*)
VAR CONSTANT
	(*Costant in lux obj*)
	NO_DIMMING	: BYTE:=0;
	DIMMING		: BYTE:=1;
	ROT			: BOOL:=1;
	GRUN		: BOOL:=0;
END_VAR

VAR_INPUT
	(* Settings *)
	ID					: WORD;
	DimmingType		: BYTE;	 (* /0: no dimming (digital), 1: dimming (analog) *)
	DimmingValForTimer	: INT;	 (* /valore 0...100 del dimming di default del lux sotto timer *)
	(* Controls *)
	CTRL_MODE			: en_Modality;	 (* 0:MAN OFF, 1:MAN-ON, 3:Timer laser, 2:Cronografo*)
	CTRL_MODE_BackUp	: en_Modality;	 (*Salvo il valore di default per il ripristino *)
	LuxTimer		: TIME; (* Tempo di accensione del lux settato nella tabella TabLuxPsg ottenuta dal file di config su SD *)
	HourMinStartOn	: TOD; (* Orario di start per rilevazione sensori start timer (Mode 03) *)
	HourMinEndOn	: TOD; (* Orario di end per rilevazione sensori start timer (Mode 03) *)
	ValInCronoInLux : INT;	(* Valore del setpoint arrivato dal crono *)
	RefTableAutLuxPsg : WORD; (* indice di riferimento alla tabella AUT_LUX_PSG se mode = 3 *)
	RestoreKey		: BOOL; (* se attivato viene ripristinato il mode di default *)
	CtrlTrig		: BOOL; (* Trigger for timer start *)
	CtrlKeyList		: ARRAY [0..9] OF BOOL; (* External KEY control input *)
	KeyQty			: BYTE; (* numero di key all'ingresso *)
	KeyMode			: en_KeyMode;	(* BYTE; //Modalità di funzionamento richiesta dal key *)
	DimmingValForKeyList: ARRAY [0..9] OF INT;
	DimmingValForKeyMax: BOOL; (* Se TRUE --> si sceglie il valore massimo; Se FALSE --> si sceglie il valore minimo *)
	ActionKey		: en_ActionKey; (* 00-NormalMode, 01-SwitchON, 02-SwitchOFF, 03-Restore *)
	(* Physical inputs *)
	Lux_State		: BOOL; (* Status feedback *)
	Lux_StateAnalog	: WORD;  (* feedback analogico dal campo GIURE ver 008  *)

END_VAR
VAR_IN_OUT
	LocalWorkingTime		: DWORD; (* [sec] Internal working time counter *)
	LocalPowerOnCycles		: WORD;	(* DWORD; Internal counter of power-on cycles *)
	LocalEnergyCounter		: WORD;	(* DWORD;  [E-1 kWh] Internal energy counter *)
	LocalEnergyCounter_t 	: DWORD; (* Temporary energy in E-2*Wsec *)
END_VAR
VAR_OUTPUT
	(* Physical outputs *)
	LuxDigitalOut	: BOOL;
	LuxAnalogOut	: WORD;
	LuxTypeOut		: BOOL;
	Lux_Enable		: BOOL;	(*  uscita logica per compatibilità con sw preesistente (ex (* Control output *)) *)
	Lux_EnableAnalog : WORD;
	(* Status *)
	Status_Log		: BYTE;
	Status_Vis 		: DWORD;
END_VAR
VAR
	TickTimer		: TON := ( PT:=T#1S );
	TrigTimer		: TOF ;

	KeyTimer		: TIME := T#200ms;
	sLux_EN			: FLT_EVENT;
	chkLux_ST		: FLT_TIME := ( TTAP:=T#20S, INITEV:=FALSE );
	chkLux_ST_Analog: FLT_TIME := ( TTAP:=T#20S, INITEV:=FALSE );
	HourMinNow		: STRING;
	semaphore		: BOOL:=GRUN;
	OnFromKey		: BOOL;
	fTrigFun		: F_TRIG;
	rTrigFun		: R_TRIG;
	fTrigKey		: F_TRIG;
	ActionKeyState	: en_ActionKey;
	KeyCounter, x	: BYTE;
	CtrlKey			: BOOL;
	DimmingValForKey: INT; (* valore 0...100 del dimming di default del lux sotto key *)
	ModeToServer : BYTE;
	ForcedOn : BYTE;
	ForcedOff : BYTE;

END_VAR
(* Con l'ID si identifica il numero del lux sul campo quindi il suo valore può variare da 1 a LUXM_MAX (attualmente 1...900) *)
IF (KeyMode = BUTTON_NO) OR (KeyMode = BUTTON_NC) THEN (* se si usano dei pulsanti sui vari digital input...*)
	KeyCounter := 0;
	FOR x:=0 TO  KeyQty-1 DO
		IF CtrlKeyList[x] = 1 THEN
			KeyCounter := KeyCounter + 1;
		END_IF
	END_FOR
	IF (KeyCounter MOD 2) = 0 THEN
		CtrlKey := FALSE;
	ELSE
		DimmingValForKey := DimmingValForKeyList[0]; (* In caso di pulsanti si prende il valore della posizione 0 dell'array *)
		CtrlKey := TRUE;
	END_IF
ELSE (* altrimenti se uso l'interruttore ne posso usare solo 1 nella posizione 0 dell'array *)
	IF (DimmingValForKeyMax) THEN
		DimmingValForKey := 0;
		FOR x:=0 TO  KeyQty-1 DO
			IF (CtrlKeyList[x] = 1) AND (DimmingValForKeyList[x] > DimmingValForKey)
			THEN
				DimmingValForKey := DimmingValForKeyList[x];
			END_IF
		END_FOR
	ELSIF NOT(DimmingValForKeyMax) THEN
		DimmingValForKey :=1000;
		FOR x:=0 TO  KeyQty-1 DO
			IF (CtrlKeyList[x] = 1) AND (DimmingValForKeyList[x] < DimmingValForKey)
			THEN
				DimmingValForKey := DimmingValForKeyList[x];
			END_IF
		END_FOR
	END_IF
	CtrlKey := 0;
	FOR x:=0 TO  KeyQty-1 DO
			CtrlKey := CtrlKey OR CtrlKeyList[x];
	END_FOR

END_IF

CASE DimmingType OF (* set dell' AsiTypeOut per sapere se eseguire il set di un analog out o di un digital out *)
	NO_DIMMING:	(* if no dimming we are using a digital output *)
		LuxTypeOut := DIGITAL; (* Set digital out mode *)
	DIMMING:	(*  if dimming we are using analog output *)
		LuxTypeOut := ANALOG; (* Set analog out mode *)
END_CASE

(* Control logic *)
(* Restore mode and value	*)
IF RestoreKey THEN
	CTRL_MODE := CTRL_MODE_BackUp;
END_IF

CASE CTRL_MODE OF
	ManualeOff: (*  0 Manuale Off *)
		(* Se commutazione arrivata da key durante funzionamento in timer o cronografo *)
		IF  NOT(CtrlKey) AND (ActionKey > NormalMode) AND ( ActionKeyState = SwitchOFF)THEN
			ActionKeyState := NormalMode;
			CTRL_MODE := CTRL_MODE_BackUp;
		ELSE
			CASE DimmingType OF
				NO_DIMMING:	(* if no dimming we are using a digital output *)
					LuxDigitalOut := TRUE; (* Lux spento (digital) *)
				DIMMING:	(*  if dimming we are using analog and digital output *)
					DimmerCtrl(); (* In caso di switch off in manuale è sempre zero anche se arriva da key *)
			END_CASE
		END_IF
	ManualeOn: (*  1 Manuale On *)
		(* Se commutazione arrivata da key durante funzionamento in timer o cronografo *)
		IF  NOT(CtrlKey) AND (ActionKey > NormalMode) AND ( ActionKeyState = SwitchON) THEN
			ActionKeyState := NormalMode;
			CTRL_MODE := CTRL_MODE_BackUp;
		ELSE
			CASE DimmingType OF
				NO_DIMMING:	(* if no dimming we are using a digital output *)
					LuxDigitalOut := FALSE; (* Lux acceso (digital) *)
				DIMMING:	(*  if dimming we are using analog and digital output  *)
					IF ActionKeyState = SwitchON THEN
						DimmerCtrlKeyOn(); (* Se il manuale on è settato a causa di un key si impongono i dati del key stesso *)
					ELSE
						DimmerCtrl();
					END_IF
			END_CASE
		END_IF
	Cronografo: (*  2 Cronografo *)
		IF  (CtrlKey) AND (ActionKey > NormalMode) THEN
			CASE  ActionKey OF
				SwitchON: 	(* Corrisponde al manuale ON *)
					CTRL_MODE := ManualeOn;
					ActionKeyState := SwitchON;
					CASE DimmingType OF
						NO_DIMMING:	(* if no dimming we are using a digital output *)
							LuxDigitalOut := FALSE; (* Lux acceso (digital) *)
						DIMMING:	(*  if dimming we are using analog and digital output  *)
							DimmerCtrlKeyOn();
					END_CASE

				SwitchOFF:	(* Corrisponde al manuale OFF  *)
					CTRL_MODE := ManualeOff;
					ActionKeyState := SwitchOFF;
					CASE DimmingType OF
						NO_DIMMING:	(* if no dimming we are using a digital output  *)
							LuxDigitalOut := TRUE; (* Lux spento (digital)  *)
						DIMMING:	(*  if dimming we are using analog and digital output  *)
							DimmerCtrlKeyOff();
					END_CASE
			END_CASE
		ELSE
			CASE DimmingType OF
				NO_DIMMING:	(* if no dimming we are using a digital output  *)
					IF ValInCronoInLux = 1000 (* OR ( LuxElement[i].PressKeyVisuOn)  *)
						THEN
						LuxDigitalOut := FALSE; (* Lux acceso (digital)  *)
						ELSE IF ValInCronoInLux = 0 (* OR ( NOT LuxElement[i].PressKeyVisuOn)  *)
							THEN
							LuxDigitalOut := TRUE; (* Lux spento (digital)  *)
						END_IF
					END_IF
				DIMMING:	(*  if dimming we are using analog output  *)
					DimmerCtrl();
			END_CASE
		END_IF
	Timer: (*  3 Timer   *)
	IF  (CtrlKey) AND (ActionKey > NormalMode) THEN
		CASE  ActionKey OF
			SwitchON: 	(* Corrisponde al manuale ON  *)
				CTRL_MODE := ManualeOn;
				ActionKeyState := SwitchON;
				CASE DimmingType OF
					NO_DIMMING:	(* if no dimming we are using a digital output  *)
						LuxDigitalOut := FALSE; (* Lux acceso (digital)  *)
					DIMMING:	(*  if dimming we are using analog and digital output   *)
						DimmerCtrlKeyOn();
				END_CASE

			SwitchOFF:	(* Corrisponde al manuale OFF  *)
				CTRL_MODE := ManualeOff;
				ActionKeyState := SwitchOFF;
				CASE DimmingType OF
					NO_DIMMING:	(* if no dimming we are using a digital output  *)
						LuxDigitalOut := TRUE; (* Lux spento (digital)  *)
					DIMMING:	(*  if dimming we are using analog and digital output  *)
						DimmerCtrlKeyOff();
				END_CASE
		END_CASE
	ELSE
		CASE DimmingType OF
			NO_DIMMING:	(* if no dimming we are using a digital output  *)
				HourMinNow:=CONCAT('TOD#', BYTE_TO_STRING(Sys.Time_Hour));
				HourMinNow:=CONCAT(HourMinNow, ':');
				HourMinNow:=CONCAT(HourMinNow, BYTE_TO_STRING(Sys.Time_Min));
				HourMinNow:=CONCAT(HourMinNow,':00');

				(* Trig timer *)
				TrigTimer.PT:=LuxTimer;
				TrigTimer(IN:= CtrlTrig);

				IF (((STRING_TO_TOD(HourMinNow) > HourMinStartOn) AND (STRING_TO_TOD(HourMinNow) < HourMinEndOn))  (* Se siamo nell'orario corretto  *)
				OR ((LuxDigitalOut = FALSE) AND (TrigTimer.Q = FALSE))) (* oppure si era acceso e adesso siamo passati fuori orario e dobbiamo spegnere  *)
				THEN
					IF TrigTimer.Q THEN
						LuxDigitalOut := FALSE; (* Lux acceso (digital)  *)
						ELSE
							LuxDigitalOut:= TRUE; (* Lux spento (digital)  *)
					END_IF
				END_IF
			DIMMING:	(*  if dimming we are using analog output  *)

				HourMinNow:=CONCAT('TOD#', BYTE_TO_STRING(Sys.Time_Hour));
				HourMinNow:=CONCAT(HourMinNow, ':');
				HourMinNow:=CONCAT(HourMinNow, BYTE_TO_STRING(Sys.Time_Min));
				HourMinNow:=CONCAT(HourMinNow,':00');

				(* Trig timer *)
				TrigTimer.PT:=LuxTimer;
				TrigTimer(IN:= CtrlTrig);

				IF (((STRING_TO_TOD(HourMinNow) > HourMinStartOn) AND (STRING_TO_TOD(HourMinNow) < HourMinEndOn))  (* Se siamo nell'orario corretto  *)
				OR ((LuxDigitalOut = FALSE) AND (TrigTimer.Q = FALSE))) (* oppure si era acceso e adesso siamo passati fuori orario e dobbiamo spegnere  *)
				THEN
					IF TrigTimer.Q THEN
						DimmerCtrl(); (* Lux acceso  *)
						ELSE
							LuxAnalogOut := 0; (* Lux spento  *)
							LuxDigitalOut := TRUE; (* Lux spento (digital)  *)
					END_IF
				END_IF
		END_CASE
		END_IF
	KeyControl: (*  4 Key function  *)
		IF CtrlKey THEN
			CASE DimmingType OF
				NO_DIMMING:	(* if no dimming we are using a digital output  *)
					LuxDigitalOut := FALSE; (* Lux acceso (digital)  *)
				DIMMING:	(*  if dimming we are using analog and digital output   *)
					DimmerCtrlKeyOn();
			END_CASE
		ELSIF CtrlKey = 0 THEN
			CASE DimmingType OF
				NO_DIMMING:	(* if no dimming we are using a digital output  *)
					LuxDigitalOut := TRUE; (* Lux spento (digital)  *)
				DIMMING:	(*  if dimming we are using analog and digital output  *)
					DimmerCtrlKeyOff();
			END_CASE
		END_IF
	END_CASE

(* ----------------------------------------------------------------------------------------------------------------------------------------  *)
(* Se i pin del feedback relè non sono cavallottati si usa la seguente riga al posto di quelle successive indicate da(#)  *)
(* REL_ST := LUX_ST[ID];	  																					 *)
(* ----------------------------------------------------------------------------------------------------------------------------------------   *)

(* setting della variabile REL_EN per compatibilità con il sw preesistente  *)
CASE DimmingType OF
	NO_DIMMING:	(* if no dimming we are using a digital output  *)
	IF LuxDigitalOut = TRUE  (* Lux spento  *)
		THEN
			(* Lux_State := FALSE;	//A causa del cavallotto sui pin del relè forzo a falso (#)  *)
			(* Lux_State := LUX_ST[ID];	  *)
			Lux_Enable := FALSE;
		ELSIF LuxDigitalOut = FALSE  (* Lux acceso			   *)
			THEN
				(* Lux_State := LUX_ST[ID];	//Quando so che la luce è accesa leggo lo stato del pin (che essendo cavallottato sarà a 1) (#)  *)
				Lux_Enable := TRUE;
	END_IF

	DIMMING:	(*  if dimming we are using analog output  *)
	IF LuxAnalogOut  = 0 (* Lux spento				  *)
		THEN
			(* REL_ST := FALSE;	 A causa del cavallotto sui pin del relè forzo a falso (#)  *)
			(* Lux_State := LUX_ST[ID];	  *)
			Lux_State:= TRUE;	(* aggiunta perchè non ho feedback sul relè *)
			Lux_Enable := FALSE;
			Lux_EnableAnalog := LuxAnalogOut; (* GIURE ver 008   *)
		ELSIF LuxAnalogOut > 0  (* Lux acceso			  *)
			THEN
				(* Lux_State := LUX_ST[ID];	 Quando so che la luce è accesa leggo lo stato del pin (che essendo cavallottato sarà a 1) (#)  *)
				Lux_State:= TRUE; (* aggiunta perchè non ho feedback sul relè *)
				Lux_Enable := TRUE;
				Lux_EnableAnalog := LuxAnalogOut;  (* GIURE ver 008  *)
	END_IF

END_CASE
(* Temporary energy counter *)
TickTimer(IN:=NOT TickTimer.Q);
IF TickTimer.Q AND Lux_Enable THEN
	LocalWorkingTime:=LocalWorkingTime+1;
	IF LocalEnergyCounter_t>36000000 THEN
		LocalEnergyCounter_t:=LocalEnergyCounter_t-36000000;
		LocalEnergyCounter:=LocalEnergyCounter+1;
	END_IF
END_IF

(* Generate status events *)
sLux_EN(IN:=Lux_Enable);
IF sLux_EN.EVL THEN
	LogEv(EL_Log,EO_LUX,ID,2,'Light OFF'); (* Light OFF  *)
END_IF
IF sLux_EN.EVH THEN
	LogEv(EL_Log,EO_LUX,ID,3,'Light ON'); (* Light ON  *)
	LocalPowerOnCycles:=LocalPowerOnCycles+1;
END_IF


(* Check status feedback *) (* GIURE ver 008 - aggiunta controllo valori analogici  *)
chkLux_ST_Analog(IN:=(Lux_StateAnalog<>Lux_EnableAnalog));
IF chkLux_ST_Analog.EVH THEN
	LogEv(EL_Alarm,EO_LUX,ID,9,'Fail Analog');(*  Feedback failure - Lux_StateAnalog<>Lux_EnableAnalog*)
END_IF
IF chkLux_ST_Analog.EVL THEN
	LogEv(EL_Log,EO_LUX,ID,1,'Successful Analog'); (*  Light feedback OK - Lux_StateAnalog = Lux_EnableAnalog  *)
END_IF
(* Check status feedback *)
chkLux_ST(IN:=(Lux_State<>Lux_Enable));
IF chkLux_ST.EVH THEN
	LogEv(EL_Alarm,EO_LUX,ID,9,'Fail'); (*  Feedback failure - Lux_State<>Lux_Enable  *)
END_IF
IF chkLux_ST.EVL THEN
	LogEv(EL_Log,EO_LUX,ID,1,'Successful'); (*  Light feedback OK - Lux_State = Lux_Enable  *)
END_IF


(* Status color *)
IF chkLux_ST.OUT THEN
	Status_Log:=2; Status_Vis:=COLOR_RED;
ELSE
	Status_Log:=0;
	Status_Vis:=SEL(Lux_Enable,COLOR_GREEN_OFF,COLOR_GREEN);
END_IF

(* Salvataggio dati in array ordinato per numero di ID utile per la visualizzazione  *)
DataLuxForVis[ID].VisStatus:=Status_Vis;
DataLuxForVis[ID].VisTimer:=LuxTimer/1000;
DataLuxForVis[ID].VisMod:=CTRL_MODE;
(* DataLuxForVis[ID].VisMod:=any_num_to_byte(CTRL_MODE); *)
END_FUNCTION_BLOCK
ACTION AddLogData:
Logger.s1:=INSERT('&LUX=',WORD_TO_STRING(ID),4);
IF ID<10 THEN Logger.s1:=INSERT(Logger.s1,'0',4); END_IF

Logger.s1:=CONCAT(Logger.s1,BOOL_TO_STRING(Lux_Enable));				Logger.s1:=CONCAT(Logger.s1,';');
Logger.s1:=CONCAT(Logger.s1,DWORD_TO_STRING(LocalWorkingTime));		Logger.s1:=CONCAT(Logger.s1,';');
Logger.s1:=CONCAT(Logger.s1,DWORD_TO_STRING(LocalPowerOnCycles));	Logger.s1:=CONCAT(Logger.s1,';');

CASE CTRL_MODE OF		(* modifica GIURE 009 ver 1.3 *)
	0: 	(*  Manuale OFF *)
		ModeToServer := 0;
		ForcedOn := 0;
		ForcedOff := 1;
	1:	(*  Manuale ON *)
		ModeToServer := 1;
		ForcedOn := 1;
		ForcedOff := 0;
	2:	(*  Cronografo *)
		ModeToServer := 2;
		ForcedOn := 0;
		ForcedOff := 0;
	3: 	(* Timer *)
		ModeToServer := 3;
		ForcedOn := 0;
		ForcedOff := 0;
END_CASE
Logger.s1:=CONCAT(Logger.s1,BYTE_TO_STRING(ModeToServer));			Logger.s1:=CONCAT(Logger.s1,';');
Logger.s1:=CONCAT(Logger.s1,BYTE_TO_STRING(Status_Log));				Logger.s1:=CONCAT(Logger.s1,';');
Logger.s1:=CONCAT(Logger.s1,BYTE_TO_STRING(ForcedOn));				Logger.s1:=CONCAT(Logger.s1,';');
Logger.s1:=CONCAT(Logger.s1,BYTE_TO_STRING(ForcedOff));				Logger.s1:=CONCAT(Logger.s1,';');
Logger.s1:=CONCAT(Logger.s1,BYTE_TO_STRING(DimmingType));			Logger.s1:=CONCAT(Logger.s1,';');
Logger.s1:=CONCAT(Logger.s1,WORD_TO_STRING(Lux_EnableAnalog/100));

ADDSTRING(ADR(Logger.TData), ADR(Logger.s1), Logger.TLen);
END_ACTION
ACTION DimmerCtrl:
CASE CTRL_MODE OF
	0: (* Manuale Off *)
		LuxAnalogOut := 0; (* Lux spento *)
		LuxDigitalOut := TRUE; (* Lux spento (digital) *)
	1: (* Manuale On *)
		LuxAnalogOut := 10000; (* Lux acceso *)
		LuxDigitalOut := FALSE; (* Lux acceso (digital) *)
	2: (* Cronografo *)
		IF ValInCronoInLux > 0 THEN
			LuxDigitalOut := FALSE; (* Lux acceso (digital) *)
			ELSE
				LuxDigitalOut := TRUE; (* Lux spento (digital) *)
		END_IF
		LuxAnalogOut := INT_TO_WORD(ValInCronoInLux*10);
	3: (* Timer 		 *)
		IF DimmingValForTimer > 0 THEN
			LuxDigitalOut := FALSE; (* Lux acceso (digital) *)
			ELSE
				LuxDigitalOut := TRUE; (* Lux spento (digital) *)
		END_IF
		LuxAnalogOut := INT_TO_WORD(DimmingValForTimer*10);
	ELSE (* default *)
		LuxDigitalOut := FALSE; (* Lux acceso (digital) *)
		LuxAnalogOut := 10000;
END_CASE
END_ACTION
ACTION DimmerCtrlKeyOff:
LuxAnalogOut := 0; (*/Lux spento*)
LuxDigitalOut := TRUE; (*Lux spento (digital)*)
END_ACTION
ACTION DimmerCtrlKeyOn:
LuxAnalogOut := INT_TO_WORD(DimmingValForKey*10);
LuxDigitalOut := FALSE; (*Lux acceso (digital) *)
END_ACTION
ACTION StatReset:
(* Reset statistic counters *)
LocalWorkingTime:=0;
LocalPowerOnCycles:=0;
LocalEnergyCounter:=0;
END_ACTION

(* POU Plant_Objects/obj_TPV, ST *)
FUNCTION_BLOCK obj_TPV
(* === TEMPERATURE PROBE  ===
   v1.0[16/04/15] - Versioning
*)
VAR CONSTANT
	NormalEv		: BYTE := 0;
	ErrorEv			: BYTE := 1;
	WarningEv		: BYTE := 2;
END_VAR
VAR_INPUT
	(* Settings *)
	ID				: BYTE;
	TAP				: BYTE:=4;	   (* Consecutive checks filter *)
	INITEV			: BOOL:= TRUE; (* Generate init OK event *)
	IN_EMIN			: INT :=-2000; (* Low error limit *)
	IN_WMIN			: INT := -550; (* Low warning value *)
	IN_WMAX			: INT :=  900; (* High warning value *)
	IN_EMAX			: INT := 8500; (* High error limit *)
	ERR_MIN_SHORT	: BOOL:= TRUE; (* TRUE  ==> EMIN=Short        , EMAX=Disconnected
									  FALSE ==> EMIN=Disconnected , EMAX=Short 		 *)
	(* Physical input *)
	IN			: INT;
END_VAR
VAR_OUTPUT
	WRN			: BOOL;	(* Value in warning range *)
	ERR			: BOOL;	(* Value error *)
	HI			: INT;	(* Highest value - cleared by Stat_Reset() action *)
	AVG			: INT; 	(* Average value - updated by Mean() action, cleared by Mean_Reset() action *)
	LOW			: INT;	(* Lowest value  - cleared by Stat_Reset() action *)

	Status_Log	: WORD;
	Status_Vis	: DWORD;
END_VAR
VAR
	cnt			: BYTE;
	event		: BYTE := 0;	(* 0: monitoring a generic, 1: monitoring an error, 2: monitoring a warning *)
	asum		: DINT;
	acnt		: WORD;
END_VAR
(* Check probe value limits *)
IF IN<=IN_EMIN OR IN>=IN_EMAX THEN
	IF NOT ERR THEN
		IF event <> ErrorEv THEN
			cnt := 1;
			event := ErrorEv;
		ELSE
			cnt:=cnt+1;
		END_IF

		IF cnt>TAP THEN
			cnt:=0;
			ERR:=TRUE; WRN:=FALSE;
			IF ( ERR_MIN_SHORT=TRUE  AND IN<=IN_EMIN ) OR ( ERR_MIN_SHORT=FALSE AND IN>=IN_EMAX ) THEN
				LogEv(EL_Alarm,EO_TPV,ID,5,INT_TO_STRING(IN));
			ELSE
				LogEv(EL_Alarm,EO_TPV,ID,4,INT_TO_STRING(IN));
			END_IF
		END_IF
	END_IF
ELSIF IN<=IN_WMIN OR IN>=IN_WMAX THEN
	IF NOT WRN THEN
		IF event <> WarningEv THEN
			cnt := 1;
			event := WarningEv;
		ELSE
			cnt:=cnt+1;
		END_IF

		IF cnt>TAP THEN
			cnt:=0;
			ERR:=FALSE; WRN:=TRUE;
			LogEv(EL_Wrn,EO_TPV,ID,SEL(IN<=IN_WMIN,3,2),INT_TO_STRING(IN));
		END_IF
	END_IF
ELSE
	IF INITEV OR WRN OR ERR THEN
		IF event <> NormalEv THEN
			cnt := 1;
			event := NormalEv;
		ELSE
			cnt:=cnt+1;
		END_IF

		IF cnt>TAP THEN
			cnt:=0;
			INITEV:=FALSE; ERR:=FALSE; WRN:=FALSE;
			LogEv(EL_Log,EO_TPV,ID,1,'Probe_OK');
		END_IF
	END_IF
END_IF


(*
(* Average value *)
IF acnt>=500 THEN
	Mean();
	asum := asum - AVG;
	acnt := acnt - 1;
END_IF

asum := asum + IN;
acnt := acnt + 1;
*)

AVG := IN;



(* Statistics values *)
IF IN<LOW THEN LOW:=IN; END_IF
IF IN>HI  THEN HI :=IN; END_IF

Lamp.obj_Status := Status_Log;
Lamp.UpdateStatus();

(* Status Log *)
IF ERR THEN	Status_Log := 2; Status_Vis := COLOR_RED;
ELSIF WRN THEN Status_Log := 1;	Status_Vis := COLOR_YELLOW;
ELSE Status_Log := 0; Status_Vis := COLOR_GREEN;
END_IF
END_FUNCTION_BLOCK
ACTION AddLogData:
Logger.s1:=INSERT('&TPV=',BYTE_TO_STRING(ID),4);
IF ID<10 THEN Logger.s1:=INSERT(Logger.s1,'0',4); END_IF
(*
Mean();
*)
Logger.s1:=CONCAT(Logger.s1,INT_TO_STRING(AVG));		Logger.s1:=CONCAT(Logger.s1,';');

Logger.s1:=CONCAT(Logger.s1,WORD_TO_STRING(Status_Log));
ADDSTRING(ADR(Logger.TData), ADR(Logger.s1), Logger.TLen);
END_ACTION
ACTION Mean:
(*AVG := DINT_TO_INT(asum/acnt); *)


AVG := IN;
END_ACTION
ACTION Mean_Reset:
AVG:=IN;
asum:=IN;
acnt:=1;
END_ACTION
ACTION Stat_Reset:
HI:=IN;
LOW:=IN;
END_ACTION

(* POU Plant_Objects/obj_VRD_new, ST *)
FUNCTION_BLOCK obj_VRD_new
(* === VALVOLA RIPARTITORE ===
   v1.0[16/04/15] - Versioning
*)
VAR CONSTANT
	Chk_CntSecAlarm	: INT := 900;	(* 900s = 15 minutes -> Observation itme *)
END_VAR
VAR_INPUT
	(* Settings *)
	ID				: BYTE;
	(* Controls *)
	RUN  			: BOOL;					(* Control input *)
	ReducedRange	: BOOL := FALSE;		(* If true output value is among 2 and 10V, otherwise 0-10V *)

	(* Physical inputs *)
	TEMP 			: INT;		(* Input temperature from sensor *)
	STATUS 			: WORD;		(* Input position from valve *)

	InitOK			: BOOL;
	Alarm1			: BOOL;
	Alarm2			: BOOL;
	Warning			: BOOL;

	Ctrl_Init		: BOOL;
	Ctrl_SetPoint	: INT;
	Ctrl_SetPointNew: INT := 0;
	Delta_SetPoint	: INT;
	Ctrl_Err		: INT;			(* Current error *)
	Ctrl_Err0		: INT; 			(* Previous error *)
	Ctrl_Accel		: REAL;			(* Derivate of error *)
	Ctrl_AccelGate  : INT:=1;		(* Derivate gate *)
	Ctrl_AccelTmr	: WORD;
	Ctrl_SetPointGate: INT := 5;	(* Setpoint gate - 0.5°C *)
	Ctrl_ErrGate	: INT:=5;		(* Error gate *)
	Ctrl_Kp			: REAL:=2;(*1;*)		(* Proportional factor *)
	Ctrl_Kd			: REAL:=10;(*100;*)  	(* Derivative factor *)
	Ctrl_Out		: REAL;

	Chk_Err			: INT;
	Chk_ErrGate		: INT:=1000; 		(* Check error gate *)
	Chk_Cnt			: INT;
	Chk_CntAlarm	: INT:=240; 		(* Check error trigger 120s *)

	(* Status *)
	Log_AvgTemp		: AVERAGE_T;
	Status_Log		: BYTE;
	Status_Vis 		: DWORD;

	(* Feedback *)
	fFeedback		: BOOL;			(* TRUE: Feedback available, FALSE: Feedback not available *)

	OffsetBoost: INT;

END_VAR
VAR_IN_OUT
(*	CLIM		: typ_Clima;  *)
END_VAR
VAR_OUTPUT
	(* Physical outputs *)
	OUT			: WORD;
END_VAR
VAR
	Curve		: CHARCURVE;
	Curve_Err	: BYTE;

	aTemp		: ARRAY [1..20] OF INT;
	meanTemp	: INT;
	sum			: INT := 0;
	Tmr			: TON := (PT:=T#1s);
	index		: BYTE;
	i			: BYTE;
	fCtrl_Err	: BOOL;		(* TRUE: Ctrl_Err>0, FALSE: Ctrl_Err<0 *)

	TON_AllarmeOvertemperatura:TON;


END_VAR


VAR_INPUT RETAIN
	Local_VRD_TAlarm: INT;
END_VAR
(* Check initialization *)
(*IF NOT InitOK THEN Init(); END_IF*)

(* Check max temperature *)

TON_AllarmeOvertemperatura(IN:=TEMP>Local_VRD_TAlarm,PT:=t#20s);
IF TON_AllarmeOvertemperatura.Q THEN
	IF NOT Alarm1 THEN
		Alarm1:=TRUE;
		LogEv(EL_AlarmStop,EO_VRD,ID,3,'VRD_Overtemperature');
	END_IF
END_IF

IF (TEMP<Local_VRD_TAlarm-10) AND Alarm1  THEN
		Alarm1:=FALSE;
END_IF




(* Check climatic setup *)
IF NOT CLIM.InitOK THEN	DefaultClim(); END_IF;
(* Calculate Setpoint *)
Curve(	IN:= T_AMB,	N:= 5, P:= CLIM.Points,			(* Given the x value as input, the corresponding y value as output is returned, if it matches the crve designed by array of points *)
		OUT=> Ctrl_SetPointNew, ERR=> Curve_Err );

IF Curve_Err>0 OR Ctrl_SetPoint>Plant_VRD_TMax THEN
	Ctrl_SetPoint:=Plant_VRD_TDefault;
	IF NOT Warning THEN
		Warning:=TRUE;
		LogEv(EL_Wrn,EO_VRD,ID,2,'VRD_Climatic_Error');
	END_IF
ELSE
	Delta_SetPoint := ABS(Ctrl_SetPoint - Ctrl_SetPointNew);
	IF Delta_SetPoint>Ctrl_SetPointGate THEN Ctrl_SetPoint := Ctrl_SetPointNew; END_IF

	Warning:=FALSE;
END_IF

Ctrl_SetPoint:=Ctrl_SetPoint+OffsetBoost;


(* Execute control loop [T=500ms] *)
(* IF RUN AND (NOT Alarm1) THEN*)
IF RUN  THEN
	(* Calculate error *)
	Ctrl_Err:=Ctrl_SetPoint-TEMP;
	(* Init/restart operations *)
	IF NOT Ctrl_Init THEN
		Ctrl_Accel:=0;
		Ctrl_AccelTmr:=0;
		Ctrl_Err0:=Ctrl_Err;
		Ctrl_Out:=5000;
		Ctrl_Init:=TRUE;
	END_IF
	(* Calculate acceleration *)
	IF ABS(Ctrl_Err-Ctrl_Err0)>Ctrl_AccelGate OR Ctrl_AccelTmr>20 THEN
		Ctrl_Accel:=INT_TO_REAL(Ctrl_Err-Ctrl_Err0)/WORD_TO_REAL(1+Ctrl_AccelTmr);
		Ctrl_AccelTmr:=0;
		Ctrl_Err0:=Ctrl_Err;
	ELSE
		Ctrl_AccelTmr:=Ctrl_AccelTmr+1;
	END_IF

	(* Gate error *)
	IF ABS(Ctrl_Err)>Ctrl_ErrGate THEN
		(* Control loop *)
		Ctrl_Out:=Ctrl_Out+(Ctrl_Kp*Ctrl_Err)+(Ctrl_Kd*Ctrl_Accel);
	END_IF

	(* Limiter and Output *)
(*	Ctrl_Out:=LIMIT(0,Ctrl_Out,27000); *)
	Ctrl_Out:=LIMIT(0,Ctrl_Out,32000);

ELSE
	Ctrl_Init:=FALSE;
	Ctrl_Out:=0;
END_IF

OUT:=SEL(Alarm1,REAL_TO_WORD(Ctrl_Out),0);





(* If there is an hardware feedback (such as 0-10V, potentiometer, ...) check it otherwise try to rebuild it *)
IF fFeedback THEN CheckFeedback();
ELSE BuildFeedback();
END_IF

(* Status temp *)
(* Status color *)
   IF Alarm1 THEN Status_Log:=2; Status_Vis:=16#2020F0;
ELSIF Warning  OR Alarm2        THEN Status_Log:=1; Status_Vis:=16#20F0F0;
                       ELSE Status_Log:=0; Status_Vis:=SEL(RUN,16#006000,16#20F020);
END_IF
END_FUNCTION_BLOCK
ACTION AddLogData:
Logger.s1:=INSERT('&VRD=',BYTE_TO_STRING(ID),4);
IF ID<10 THEN Logger.s1:=INSERT(Logger.s1,'0',4); END_IF


Logger.s1:=CONCAT(Logger.s1,INT_TO_STRING(Ctrl_SetPoint));				Logger.s1:=CONCAT(Logger.s1,';');

(* gli passo la percentuale di comando che ricavo dalla divisone per 327 del comando fisico *)
Logger.s1:=CONCAT(Logger.s1,WORD_TO_STRING(OUT/327));						Logger.s1:=CONCAT(Logger.s1,';');


(* gli passo la percentuale di apertura che ricavo dalla divisone per 327 del comando fisico *)
IF fFeedback THEN Logger.s1:=CONCAT(Logger.s1,WORD_TO_STRING(STATUS/327));
ELSE Logger.s1:=CONCAT(Logger.s1,'0');	(* Bypass *)
END_IF

Logger.s1:=CONCAT(Logger.s1,';');

Logger.s1:=CONCAT(Logger.s1,WORD_TO_STRING(Status_Log));

Logger.s1:=CONCAT(Logger.s1,';');
Logger.s1:=CONCAT(Logger.s1,'1'); (* Valvola modulante controllata Analogica *)

ADDSTRING(ADR(Logger.TData), ADR(Logger.s1), Logger.TLen);
END_ACTION
ACTION BuildFeedback:
(* Comparison is taken between actual temperature vs windowed mean value of last 20 temperature
   (check is carried out every second)	*)
IF RUN AND (NOT Alarm1) THEN

	IF Ctrl_Err>0 THEN
		IF NOT fCtrl_Err THEN index := 0; END_IF
		fCtrl_Err := TRUE;
	ELSE
		IF fCtrl_Err THEN index := 0; END_IF
		fCtrl_Err := FALSE;
	END_IF

	(* Temperature is lower than setpoint -->> Should increase *)
	Tmr(IN:=NOT Tmr.Q);

	IF Tmr.Q THEN

		IF index<21 THEN
			(* Fullfil temperature array *)
			aTemp[index] := TEMP;
			index := index + 1;

			IF index=20 THEN
				FOR i:=1 TO 20 BY 1 DO sum := sum + aTemp[i]; END_FOR
			END_IF
		ELSE
			(* Calculate mean value *)
			meanTemp := sum/20;

			IF (fCtrl_Err AND TEMP<meanTemp) OR (NOT fCtrl_Err AND TEMP>meanTemp) THEN

				IF Chk_Cnt>Chk_CntSecAlarm THEN
					IF NOT Alarm2 THEN
						Alarm2:=TRUE;
						LogEv(EL_Alarm,EO_VRD,ID,4,'VRD_Position_Error');
					END_IF
				ELSE
					Chk_Cnt := Chk_Cnt+1;
				END_IF

			ELSE
				(* Reset counter and alarm flag *)
				Chk_Cnt:=0;
				Alarm2:=FALSE;
			END_IF

			sum := 0;	(* Reset sum counter *)

			(* Shift array removing oldest value *)
			FOR i:=1 TO 20 BY 1 DO
				aTemp[i-1] := aTemp[i];
				sum := sum + aTemp[i];
			END_FOR

			aTemp[20] := TEMP;			(* Last temperature value is new one *)
			sum := sum + aTemp[20];		(* Update sum *)
		END_IF
	END_IF
END_IF
END_ACTION
ACTION CheckFeedback:
(* Calculate position error according to feedback *)
IF ReducedRange THEN
(* SETPOINT[2..10V]-STATUS[0..10V] *)
	IF OUT<=6553 THEN Chk_Err:=0; ELSE Chk_Err:=(OUT-6553)/262; END_IF
	Chk_Err:=(Chk_Err-STATUS)/327;
ELSE
(* SETPOINT[0..10V]-STATUS[0..10V] *)
	Chk_Err := OUT - STATUS;
END_IF

(* Check position error *)
IF ( ABS(Chk_Err)>Chk_ErrGate ) THEN
	IF Chk_Cnt>Chk_CntAlarm THEN
		IF NOT Alarm2 THEN
			Alarm2:=TRUE;
			LogEv(EL_Wrn,EO_VRD,ID,4,'VRD_Position_Error');
		END_IF
	ELSE
		Chk_Cnt:=Chk_Cnt+1;
	END_IF
ELSE
	Chk_Cnt:=0;
	Alarm2:=FALSE;
END_IF
END_ACTION
ACTION DefaultClim:
(*CLIM.Points[0].X:=-300; CLIM.Points[0].Y:=400;
CLIM.Points[1].X:=-50;  CLIM.Points[1].Y:=400;
CLIM.Points[2].X:= 200; CLIM.Points[2].Y:=200;
CLIM.Points[3].X:= 300; CLIM.Points[3].Y:=200;
CLIM.Points[4].X:= 500; CLIM.Points[4].Y:=200;*)
CLIM.Points[0].X:=-300; CLIM.Points[0].Y:=850;
CLIM.Points[1].X:=-50;  CLIM.Points[1].Y:=650;
CLIM.Points[2].X:= 100; CLIM.Points[2].Y:=400;
CLIM.Points[3].X:= 200; CLIM.Points[3].Y:=200;
CLIM.Points[4].X:= 500; CLIM.Points[4].Y:=200;
CLIM.InitOK:=TRUE;
LogEv(EL_Wrn,EO_VRD,ID,1,'Climatic_Default');
END_ACTION
ACTION Init:
(* End initialization *)
InitOK:=TRUE;
END_ACTION

(* POU Utils Functions/PLANT_STATUS, ST *)
FUNCTION_BLOCK PLANT_STATUS
VAR_INPUT
	obj_Status		:	WORD;
END_VAR
VAR_OUTPUT
END_VAR
VAR
	PLANT_STATUS	:	WORD;

	Pwm				:	TON := (PT:=T#1s);
END_VAR
CASE plant_Status OF

	0:	(* Plant OK - Everything works well *)
		(*Pwm(IN:=FALSE);	*)						(* Stop timer if running *)
		LAMP_AL := FALSE;						(* Keep the lamp switched off *)

	(*1:	(* Plant in warning *)
		Pwm(IN:= NOT(Pwm.Q));

		IF Pwm.Q THEN
			LAMP_AL := NOT LAMP_AL;				(* Toggle output *)
		END_IF*)

	2:	(* Plant in alarm *)
		(*Pwm(IN:=FALSE);	*)						(* Stop timer if running *)
		LAMP_AL	:= TRUE;						(* Keep the lamp switched on *)

END_CASE

plant_Status := 0;		(* Reset plant status *)
END_FUNCTION_BLOCK
ACTION UpdateStatus:
IF plant_Status = 2 THEN

	RETURN;					(* If plant already in alarm condition do nothing *)

ELSE

		IF obj_Status <> 0 THEN
			plant_Status := obj_Status;			(* If plant in warning/normal condition and current object in alarm, update plant status *)
		END_IF
END_IF
END_ACTION

(* POU PLC_WDT, ST *)
FUNCTION PLC_WDT: DWORD VAR_INPUT dwEvent: DWORD; dwFilter: DWORD; dwOwner: DWORD; END_VAR
LogEv(EL_AlarmStop,EO_SYS,1,10,'Watchdog');
END_FUNCTION

(* POU Utils Functions/RAWTOHEXSTR, ST *)
FUNCTION RAWTOHEXSTR : STRING(128)
VAR_INPUT
	pData: POINTER TO BYTE;
	DataLen: BYTE;
END_VAR
VAR
	pt: POINTER TO BYTE;
	xl: BYTE;
END_VAR
pt:=ADR(RAWTOHEXSTR);

xl:=2;

WHILE DataLen>0 AND xl<128 DO

	pt^ := (pData^ / 16#10) + 48 + (((pData^ / 16#10)/10)*7);
	pt:=pt+1;
	pt^ := (pData^ AND 16#0F)  + 48 + (((pData^ AND 16#0F)/10)*7);
	pt:=pt+1;

	xl:=xl+2;

	DataLen:=DataLen-1;
	pData:=pData+1;

END_WHILE

pt^:=0;
END_FUNCTION

(* POU Utils/RTC_Update, ST *)
FUNCTION RTC_Update : BOOL
VAR
	T: DT;
	TS: STRING;
	TS2: STRING;
	Hour: BYTE;
	Minute: BYTE;
END_VAR
(* Get RTC time *)
T:=SysRtcGetTime(TRUE);
Sys.Time_CT_DT:=T;
(* Calculate variables *)
TS:=DT_TO_STRING(T);
Sys.Time_LogString:=DELETE(STR:=TS, LEN:=3, POS:=1);
TS2:=MID(STR:=TS, LEN:=4, POS:= 4); Sys.Time_Year 	:=STRING_TO_WORD(TS2);
TS2:=MID(STR:=TS, LEN:=2, POS:= 9); Sys.Time_Month	:=STRING_TO_BYTE(TS2);
TS2:=MID(STR:=TS, LEN:=2, POS:=12); Sys.Time_Day  	:=STRING_TO_BYTE(TS2);
Sys.Time_CT_Day:=(32*(Sys.Time_Month-1)+Sys.Time_Day-1);
TS2:=MID(STR:=TS, LEN:=2, POS:=15); Hour			:=STRING_TO_BYTE(TS2);
TS2:=MID(STR:=TS, LEN:=2, POS:=18); Minute		 	:=STRING_TO_BYTE(TS2);
Sys.Time_Hour := Hour;
Sys.Time_Minute := Minute;
Sys.Time_CT_Quarter:=Hour*4+(Minute/15);
Sys.Time_CT_Minute:=Hour*60+Minute;
END_FUNCTION

(* POU Utils Functions/SHIFT_ARRAY, ST *)
FUNCTION SHIFT_ARRAY : BOOL
VAR_INPUT
	pData	:	POINTER TO ARRAY [1..2] OF WORD;
	Size	:	BYTE;
END_VAR
VAR
	pNew	:	POINTER TO WORD;
	i		:	BYTE;
END_VAR
(* Shift right *)
FOR i:=1 TO (Size-1) BY 1 DO

	(*pNew := pData + 1;*)
	pData^[i] := pData^[i+1];
	(*pData := pData + 1;*)

END_FOR
END_FUNCTION

(* POU Utils Functions/TONOF, ST *)
FUNCTION_BLOCK TONOF
VAR_INPUT
	IN		: BOOL;
	PT_ON	: TIME; (* time to pass, before OUT is set *)
	PT_OF	: TIME; (* time to pass, before OUT is reset *)
END_VAR
VAR_OUTPUT
	OUT		: BOOL;
END_VAR
VAR
	timer	: TON;
END_VAR
IF IN<>OUT THEN
	timer(IN:=TRUE,PT:=SEL(IN,PT_OF,PT_ON));
	IF timer.Q THEN OUT:=IN; END_IF
ELSE
	timer(IN:=FALSE);
END_IF
END_FUNCTION_BLOCK

(* Visualisation PLC_VISU
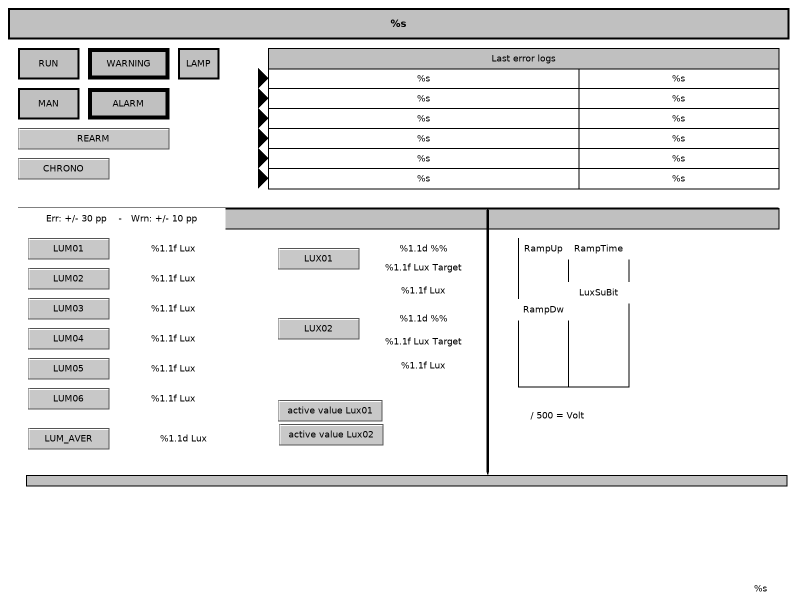
rectangle at (10,10)-(791,41): text "%s"; shows .Plant_NAME
rectangle at (530,580)-(771,601): text "%s"; shows Sys.Time_LogString
rounded rectangle at (20,50)-(81,81): text "RUN"; alarm colour if NOT Mode_Manual; runs INTERN ASSIGN Mode_Manual:=(FALSE)
rounded rectangle at (20,90)-(81,121): text "MAN"; alarm colour if Mode_Manual; runs INTERN ASSIGN Mode_Manual:=(TRUE)
rectangle at (580,70)-(781,91): text "%s"; shows Sys.LastLogs_Msg[0]
polygon at (260,170)-(270,190): invisible if Sys.LastLogs_Idx<>0
rectangle at (580,90)-(781,111): text "%s"; shows Sys.LastLogs_Msg[1]
polygon at (260,70)-(270,90): invisible if Sys.LastLogs_Idx<>1
rectangle at (580,110)-(781,131): text "%s"; shows Sys.LastLogs_Msg[2]
polygon at (260,90)-(270,110): invisible if Sys.LastLogs_Idx<>2
rectangle at (580,130)-(781,151): text "%s"; shows Sys.LastLogs_Msg[3]
polygon at (260,110)-(270,130): invisible if Sys.LastLogs_Idx<>3
rectangle at (580,150)-(781,171): text "%s"; shows Sys.LastLogs_Msg[4]
polygon at (260,130)-(270,150): invisible if Sys.LastLogs_Idx<>4
rectangle at (580,170)-(781,191): text "%s"; shows Sys.LastLogs_Msg[5]
polygon at (260,150)-(270,170): invisible if Sys.LastLogs_Idx<>5
rectangle at (270,70)-(581,91): text "%s"; shows Sys.LastLogs_Dat[0]
rectangle at (270,90)-(581,111): text "%s"; shows Sys.LastLogs_Dat[1]
rectangle at (270,110)-(581,131): text "%s"; shows Sys.LastLogs_Dat[2]
rectangle at (270,130)-(581,151): text "%s"; shows Sys.LastLogs_Dat[3]
rectangle at (270,150)-(581,171): text "%s"; shows Sys.LastLogs_Dat[4]
rectangle at (270,170)-(581,191): text "%s"; shows Sys.LastLogs_Dat[5]
rectangle at (90,90)-(171,121): text "ALARM"; alarm colour if Sys.Alarm; runs INTERN ASSIGN Mode_Manual:=(FALSE)
rectangle at (90,50)-(171,81): text "WARNING"; alarm colour if Sys.Warning; runs INTERN ASSIGN Mode_Manual:=(TRUE)
button at (20,130)-(171,151): text "REARM"; runs INTERN ASSIGN Sys.Alarm:=(FALSE);INTERN ASSIGN Sys.Warning:=(FALSE)
rectangle at (270,50)-(781,71): text "Last error logs"
rectangle at (520,240)-(571,261): text "RampUp"
rounded rectangle at (180,50)-(221,81): text "LAMP"; alarm colour if LAMP_AL
button at (20,160)-(111,181): text "CHRONO"; opens VIS_CHONOEDITOR
button at (30,240)-(111,261): text "LUM01"
rectangle at (130,240)-(221,261): text "%1.1f Lux"; shows INT_TO_REAL(LumList[1].IN)*LuxSuBit
button at (30,270)-(111,291): text "LUM02"
rectangle at (130,270)-(221,291): text "%1.1f Lux"; shows INT_TO_REAL(LumList[2].IN)*LuxSuBit
button at (30,300)-(111,321): text "LUM03"
rectangle at (130,300)-(221,321): text "%1.1f Lux"; shows INT_TO_REAL(LumList[3].IN)*LuxSuBit
button at (30,330)-(111,351): text "LUM04"
rectangle at (130,330)-(221,351): text "%1.1f Lux"; shows INT_TO_REAL(LumList[4].IN)*LuxSuBit
button at (30,360)-(111,381): text "LUM05"
rectangle at (130,360)-(221,381): text "%1.1f Lux"; shows INT_TO_REAL(LumList[5].IN)*LuxSuBit
button at (30,390)-(111,411): text "LUM06"
rectangle at (130,390)-(221,411): text "%1.1f Lux"; shows DWORD_TO_REAL(LumList[6].IN)*LuxSuBit
button at (30,430)-(111,451): text "LUM_AVER"
rectangle at (140,430)-(231,451): text "%1.1d Lux"; shows PLC_PRG.LumValueAverageLux
button at (280,250)-(361,271): text "LUX01"
rectangle at (380,240)-(471,261): text "%1.1d %%"; shows LuxOutput[1].AnalogOut/100
rectangle at (380,282)-(471,303): text "%1.1f Lux"; shows INT_TO_REAL(LUX01)*LuxSuBit
button at (280,320)-(361,341): text "LUX02"
rectangle at (380,310)-(471,331): text "%1.1d %%"; shows LuxOutput[2].AnalogOut/100
rectangle at (380,357)-(471,378): text "%1.1f Lux"; shows INT_TO_REAL(LUX02)*LuxSuBit
rectangle at (520,301)-(571,322): text "RampDw"
rectangle at (570,240)-(631,261): text "RampTime"
rectangle at (20,210)-(227,231): text "Err: +/- 30 pp    -   Wrn: +/- 10 pp"
button at (280,402)-(384,423): text "active value Lux01"; toggles PLC_PRG.ValInCronoFromVisu[1]
button at (281,426)-(385,447): text "active value Lux02"; toggles PLC_PRG.ValInCronoFromVisu[2]
rectangle at (380,333)-(471,354): text "%1.1f Lux Target"; shows LuxOutput[2].AnalogOut*3.27*LuxSuBit
rectangle at (380,259)-(471,280): text "%1.1f Lux Target"; shows LuxOutput[1].AnalogOut*3.27*LuxSuBit
rectangle at (570,284)-(631,305): text "LuxSuBit"
rectangle at (521,407)-(598,428): text "/ 500 = Volt"
7 more shapes without text or variables
18 elements of other kinds (tables, trends, ...) not read
*)

(* Visualisation VIS_CHONOEDITOR
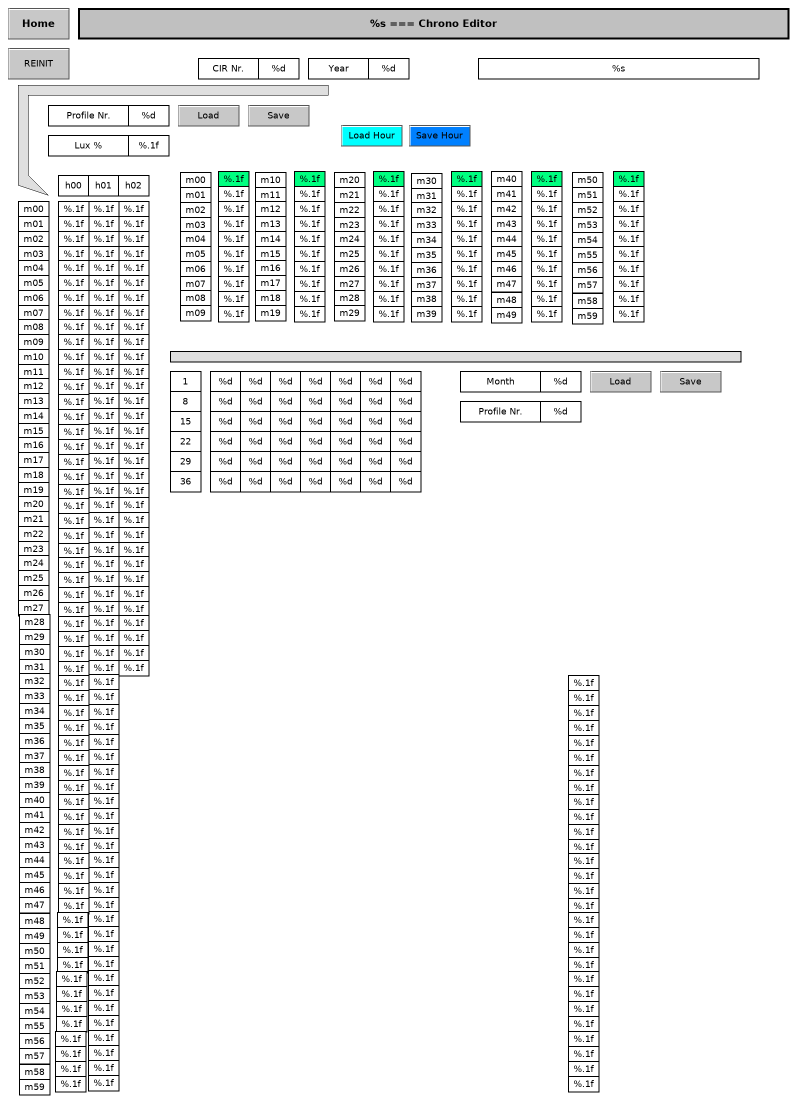
rectangle at (200,60)-(261,81): text "CIR Nr."
rectangle at (260,60)-(301,81): text "%d"; shows CronEd.CN_Sel; alarm colour if CronEd.CN_Sel<>CronEd.CN_Act; editable 1..250
rectangle at (50,107)-(131,128): text "Profile Nr."
rectangle at (130,107)-(171,128): text "%d"; shows CronEd.PR_Sel; alarm colour if CronEd.PR_Sel<>CronEd.PR_Act; editable 1..10
rectangle at (50,137)-(131,158): text "Lux %"
rectangle at (130,137)-(171,158): text "%.1f"; shows CronEd.PR_TT; editable
button at (180,107)-(241,128): text "Load"; toggles CronEd.PR_Load
button at (250,107)-(311,128): text "Save"; toggles CronEd.PR_Save
rectangle at (20,203)-(51,219): text "m00"
rectangle at (20,218)-(51,234): text "m01"
rectangle at (20,233)-(51,249): text "m02"
rectangle at (20,248)-(51,264): text "m03"
rectangle at (80,10)-(791,41): text "%s === Chrono Editor"; shows .Plant_NAME
button at (10,10)-(71,41): text "Home"; opens PLC_VISU
rectangle at (60,177)-(91,198): text "h00"; runs INTERN ASSIGN CronEd.PR.Setpoint[0]:=(REAL_TO_WORD(CronEd.PR_TT*10));INTERN ASSIGN CronEd.PR.Setpoint[1]:=(REAL_TO_WORD(CronEd.PR_TT*10));INTERN ASSIGN CronEd.PR.Setpoint[2]:=(REAL_TO_WORD(CronEd.PR_TT*10));INTERN ASSIGN CronEd.PR.Setpoint[3]:=(REAL_TO_WORD(CronEd.PR_TT*10))
rectangle at (90,177)-(121,198): text "h01"; runs INTERN ASSIGN CronEd.PR.Setpoint[4]:=(REAL_TO_WORD(CronEd.PR_TT*10));INTERN ASSIGN CronEd.PR.Setpoint[5]:=(REAL_TO_WORD(CronEd.PR_TT*10));INTERN ASSIGN CronEd.PR.Setpoint[6]:=(REAL_TO_WORD(CronEd.PR_TT*10));INTERN ASSIGN CronEd.PR.Setpoint[7]:=(REAL_TO_WORD(CronEd.PR_TT*10))
rectangle at (120,177)-(151,198): text "h02"; runs INTERN ASSIGN CronEd.PR.Setpoint[8]:=(REAL_TO_WORD(CronEd.PR_TT*10));INTERN ASSIGN CronEd.PR.Setpoint[9]:=(REAL_TO_WORD(CronEd.PR_TT*10));INTERN ASSIGN CronEd.PR.Setpoint[10]:=(REAL_TO_WORD(CronEd.PR_TT*10));INTERN ASSIGN CronEd.PR.Setpoint[11]:=(REAL_TO_WORD(CronEd.PR_TT*10))
rectangle at (462,373)-(543,394): text "Month"
rectangle at (542,373)-(583,394): text "%d"; shows CronEd.CA_Sel; alarm colour if CronEd.CA_Sel<>CronEd.CA_Act; editable 1..12
rectangle at (462,403)-(543,424): text "Profile Nr."
rectangle at (542,403)-(583,424): text "%d"; shows CronEd.CA_TPR; editable 0..10
button at (592,373)-(653,394): text "Load"; toggles CronEd.CA_Load
button at (662,373)-(723,394): text "Save"; toggles CronEd.CA_Save
rounded rectangle at (212,373)-(243,394): text "%d"; shows CronEd.CA.Profile[0]; invisible if CronEd.CA_DayF>0; alarm colour if CronEd.CA.Profile[0]=0; runs INTERN ASSIGN CronEd.CA.Profile[0]:=(CronEd.CA_TPR)
rectangle at (172,373)-(203,394): text "1"
rounded rectangle at (242,373)-(273,394): text "%d"; shows CronEd.CA.Profile[1]; invisible if CronEd.CA_DayF>1; alarm colour if CronEd.CA.Profile[1]=0; runs INTERN ASSIGN CronEd.CA.Profile[1]:=(CronEd.CA_TPR)
rounded rectangle at (272,373)-(303,394): text "%d"; shows CronEd.CA.Profile[2]; invisible if CronEd.CA_DayF>2; alarm colour if CronEd.CA.Profile[2]=0; runs INTERN ASSIGN CronEd.CA.Profile[2]:=(CronEd.CA_TPR)
rounded rectangle at (302,373)-(333,394): text "%d"; shows CronEd.CA.Profile[3]; invisible if CronEd.CA_DayF>3; alarm colour if CronEd.CA.Profile[3]=0; runs INTERN ASSIGN CronEd.CA.Profile[3]:=(CronEd.CA_TPR)
rounded rectangle at (332,373)-(363,394): text "%d"; shows CronEd.CA.Profile[4]; invisible if CronEd.CA_DayF>4; alarm colour if CronEd.CA.Profile[4]=0; runs INTERN ASSIGN CronEd.CA.Profile[4]:=(CronEd.CA_TPR)
rounded rectangle at (362,373)-(393,394): text "%d"; shows CronEd.CA.Profile[5]; invisible if CronEd.CA_DayF>5; alarm colour if CronEd.CA.Profile[5]=0; runs INTERN ASSIGN CronEd.CA.Profile[5]:=(CronEd.CA_TPR)
rounded rectangle at (392,373)-(423,394): text "%d"; shows CronEd.CA.Profile[6]; alarm colour if CronEd.CA.Profile[6]=0; runs INTERN ASSIGN CronEd.CA.Profile[6]:=(CronEd.CA_TPR)
rounded rectangle at (212,393)-(243,414): text "%d"; shows CronEd.CA.Profile[7]; alarm colour if CronEd.CA.Profile[7]=0; runs INTERN ASSIGN CronEd.CA.Profile[7]:=(CronEd.CA_TPR)
rectangle at (172,393)-(203,414): text "8"
rounded rectangle at (242,393)-(273,414): text "%d"; shows CronEd.CA.Profile[8]; alarm colour if CronEd.CA.Profile[8]=0; runs INTERN ASSIGN CronEd.CA.Profile[8]:=(CronEd.CA_TPR)
rounded rectangle at (272,393)-(303,414): text "%d"; shows CronEd.CA.Profile[9]; alarm colour if CronEd.CA.Profile[9]=0; runs INTERN ASSIGN CronEd.CA.Profile[9]:=(CronEd.CA_TPR)
rounded rectangle at (302,393)-(333,414): text "%d"; shows CronEd.CA.Profile[10]; alarm colour if CronEd.CA.Profile[10]=0; runs INTERN ASSIGN CronEd.CA.Profile[10]:=(CronEd.CA_TPR)
rounded rectangle at (332,393)-(363,414): text "%d"; shows CronEd.CA.Profile[11]; alarm colour if CronEd.CA.Profile[11]=0; runs INTERN ASSIGN CronEd.CA.Profile[11]:=(CronEd.CA_TPR)
rounded rectangle at (362,393)-(393,414): text "%d"; shows CronEd.CA.Profile[12]; alarm colour if CronEd.CA.Profile[12]=0; runs INTERN ASSIGN CronEd.CA.Profile[12]:=(CronEd.CA_TPR)
rounded rectangle at (392,393)-(423,414): text "%d"; shows CronEd.CA.Profile[13]; alarm colour if CronEd.CA.Profile[13]=0; runs INTERN ASSIGN CronEd.CA.Profile[13]:=(CronEd.CA_TPR)
rounded rectangle at (212,413)-(243,434): text "%d"; shows CronEd.CA.Profile[14]; alarm colour if CronEd.CA.Profile[14]=0; runs INTERN ASSIGN CronEd.CA.Profile[14]:=(CronEd.CA_TPR)
rectangle at (172,413)-(203,434): text "15"
rounded rectangle at (242,413)-(273,434): text "%d"; shows CronEd.CA.Profile[15]; alarm colour if CronEd.CA.Profile[15]=0; runs INTERN ASSIGN CronEd.CA.Profile[15]:=(CronEd.CA_TPR)
rounded rectangle at (272,413)-(303,434): text "%d"; shows CronEd.CA.Profile[16]; alarm colour if CronEd.CA.Profile[16]=0; runs INTERN ASSIGN CronEd.CA.Profile[16]:=(CronEd.CA_TPR)
rounded rectangle at (302,413)-(333,434): text "%d"; shows CronEd.CA.Profile[17]; alarm colour if CronEd.CA.Profile[17]=0; runs INTERN ASSIGN CronEd.CA.Profile[17]:=(CronEd.CA_TPR)
rounded rectangle at (332,413)-(363,434): text "%d"; shows CronEd.CA.Profile[18]; alarm colour if CronEd.CA.Profile[18]=0; runs INTERN ASSIGN CronEd.CA.Profile[18]:=(CronEd.CA_TPR)
rounded rectangle at (362,413)-(393,434): text "%d"; shows CronEd.CA.Profile[19]; alarm colour if CronEd.CA.Profile[19]=0; runs INTERN ASSIGN CronEd.CA.Profile[19]:=(CronEd.CA_TPR)
rounded rectangle at (392,413)-(423,434): text "%d"; shows CronEd.CA.Profile[20]; alarm colour if CronEd.CA.Profile[20]=0; runs INTERN ASSIGN CronEd.CA.Profile[20]:=(CronEd.CA_TPR)
rounded rectangle at (212,433)-(243,454): text "%d"; shows CronEd.CA.Profile[21]; alarm colour if CronEd.CA.Profile[21]=0; runs INTERN ASSIGN CronEd.CA.Profile[21]:=(CronEd.CA_TPR)
rectangle at (172,433)-(203,454): text "22"
rounded rectangle at (242,433)-(273,454): text "%d"; shows CronEd.CA.Profile[22]; alarm colour if CronEd.CA.Profile[22]=0; runs INTERN ASSIGN CronEd.CA.Profile[22]:=(CronEd.CA_TPR)
rounded rectangle at (272,433)-(303,454): text "%d"; shows CronEd.CA.Profile[23]; alarm colour if CronEd.CA.Profile[23]=0; runs INTERN ASSIGN CronEd.CA.Profile[23]:=(CronEd.CA_TPR)
rounded rectangle at (302,433)-(333,454): text "%d"; shows CronEd.CA.Profile[24]; alarm colour if CronEd.CA.Profile[24]=0; runs INTERN ASSIGN CronEd.CA.Profile[24]:=(CronEd.CA_TPR)
rounded rectangle at (332,433)-(363,454): text "%d"; shows CronEd.CA.Profile[25]; alarm colour if CronEd.CA.Profile[25]=0; runs INTERN ASSIGN CronEd.CA.Profile[25]:=(CronEd.CA_TPR)
rounded rectangle at (362,433)-(393,454): text "%d"; shows CronEd.CA.Profile[26]; alarm colour if CronEd.CA.Profile[26]=0; runs INTERN ASSIGN CronEd.CA.Profile[26]:=(CronEd.CA_TPR)
rounded rectangle at (392,433)-(423,454): text "%d"; shows CronEd.CA.Profile[27]; alarm colour if CronEd.CA.Profile[27]=0; runs INTERN ASSIGN CronEd.CA.Profile[27]:=(CronEd.CA_TPR)
rounded rectangle at (212,453)-(243,474): text "%d"; shows CronEd.CA.Profile[28]; alarm colour if CronEd.CA.Profile[28]=0; runs INTERN ASSIGN CronEd.CA.Profile[28]:=(CronEd.CA_TPR)
rectangle at (172,453)-(203,474): text "29"
rounded rectangle at (242,453)-(273,474): text "%d"; shows CronEd.CA.Profile[29]; alarm colour if CronEd.CA.Profile[29]=0; runs INTERN ASSIGN CronEd.CA.Profile[29]:=(CronEd.CA_TPR)
rounded rectangle at (272,453)-(303,474): text "%d"; shows CronEd.CA.Profile[30]; alarm colour if CronEd.CA.Profile[30]=0; runs INTERN ASSIGN CronEd.CA.Profile[30]:=(CronEd.CA_TPR)
rounded rectangle at (302,453)-(333,474): text "%d"; shows CronEd.CA.Profile[31]; alarm colour if CronEd.CA.Profile[31]=0; runs INTERN ASSIGN CronEd.CA.Profile[31]:=(CronEd.CA_TPR)
rounded rectangle at (332,453)-(363,474): text "%d"; shows CronEd.CA.Profile[32]; invisible if CronEd.CA_DayL<32; alarm colour if CronEd.CA.Profile[32]=0; runs INTERN ASSIGN CronEd.CA.Profile[32]:=(CronEd.CA_TPR)
rounded rectangle at (362,453)-(393,474): text "%d"; shows CronEd.CA.Profile[33]; invisible if CronEd.CA_DayL<33; alarm colour if CronEd.CA.Profile[33]=0; runs INTERN ASSIGN CronEd.CA.Profile[33]:=(CronEd.CA_TPR)
rounded rectangle at (392,453)-(423,474): text "%d"; shows CronEd.CA.Profile[34]; invisible if CronEd.CA_DayL<34; alarm colour if CronEd.CA.Profile[34]=0; runs INTERN ASSIGN CronEd.CA.Profile[34]:=(CronEd.CA_TPR)
rounded rectangle at (212,473)-(243,494): text "%d"; shows CronEd.CA.Profile[35]; invisible if CronEd.CA_DayL<35; alarm colour if CronEd.CA.Profile[35]=0; runs INTERN ASSIGN CronEd.CA.Profile[35]:=(CronEd.CA_TPR)
rectangle at (172,473)-(203,494): text "36"; invisible if CronEd.CA_DayL<35
rounded rectangle at (242,473)-(273,494): text "%d"; shows CronEd.CA.Profile[36]; invisible if CronEd.CA_DayL<36; alarm colour if CronEd.CA.Profile[36]=0; runs INTERN ASSIGN CronEd.CA.Profile[36]:=(CronEd.CA_TPR)
rounded rectangle at (272,473)-(303,494): text "%d"; shows CronEd.CA.Profile[37]; invisible if CronEd.CA_DayL<37; alarm colour if CronEd.CA.Profile[37]=0; runs INTERN ASSIGN CronEd.CA.Profile[37]:=(CronEd.CA_TPR)
rounded rectangle at (302,473)-(333,494): text "%d"; shows CronEd.CA.Profile[38]; invisible if CronEd.CA_DayL<38; alarm colour if CronEd.CA.Profile[38]=0; runs INTERN ASSIGN CronEd.CA.Profile[38]:=(CronEd.CA_TPR)
rounded rectangle at (332,473)-(363,494): text "%d"; shows CronEd.CA.Profile[39]; invisible if CronEd.CA_DayL<39; alarm colour if CronEd.CA.Profile[39]=0; runs INTERN ASSIGN CronEd.CA.Profile[39]:=(CronEd.CA_TPR)
rounded rectangle at (362,473)-(393,494): text "%d"; shows CronEd.CA.Profile[40]; invisible if CronEd.CA_DayL<40; alarm colour if CronEd.CA.Profile[40]=0; runs INTERN ASSIGN CronEd.CA.Profile[40]:=(CronEd.CA_TPR)
rounded rectangle at (392,473)-(423,494): text "%d"; shows CronEd.CA.Profile[41]; invisible if CronEd.CA_DayL<41; alarm colour if CronEd.CA.Profile[41]=0; runs INTERN ASSIGN CronEd.CA.Profile[41]:=(CronEd.CA_TPR)
rectangle at (310,60)-(371,81): text "Year"
rectangle at (370,60)-(411,81): text "%d"; shows CronEd.CN_YSel; alarm colour if CronEd.CN_YSel<>CronEd.CN_YAct; editable 2000..2100
rectangle at (480,60)-(761,81): text "%s"; shows CronEd.Message
button at (10,50)-(71,81): text "REINIT"; runs INTERN ASSIGN CRON[1].InitOK:=(FALSE);INTERN ASSIGN CRON[2].InitOK:=(FALSE)
rectangle at (20,262)-(51,278): text "m04"
rectangle at (20,277)-(51,293): text "m05"
rectangle at (20,292)-(51,308): text "m06"
rectangle at (20,307)-(51,323): text "m07"
rectangle at (20,321)-(51,337): text "m08"
rectangle at (20,336)-(51,352): text "m09"
rectangle at (20,351)-(51,367): text "m10"
rectangle at (20,366)-(51,382): text "m11"
rectangle at (20,380)-(51,396): text "m12"
rectangle at (20,395)-(51,411): text "m13"
rectangle at (20,410)-(51,426): text "m14"
rectangle at (20,425)-(51,441): text "m15"
rectangle at (20,439)-(51,455): text "m16"
rectangle at (20,454)-(51,470): text "m17"
rectangle at (20,469)-(51,485): text "m18"
rectangle at (20,484)-(51,500): text "m19"
rounded rectangle at (120,203)-(151,219): text "%.1f"; shows WORD_TO_REAL(CronEd.PR.Setpoint[120])/10; runs INTERN ASSIGN CronEd.PR.Setpoint[120]:=(REAL_TO_WORD(CronEd.PR_TT*10))
rounded rectangle at (120,218)-(151,234): text "%.1f"; shows WORD_TO_REAL(CronEd.PR.Setpoint[121])/10; runs INTERN ASSIGN CronEd.PR.Setpoint[121]:=(REAL_TO_WORD(CronEd.PR_TT*10))
rounded rectangle at (120,233)-(151,249): text "%.1f"; shows WORD_TO_REAL(CronEd.PR.Setpoint[122])/10; runs INTERN ASSIGN CronEd.PR.Setpoint[122]:=(REAL_TO_WORD(CronEd.PR_TT*10))
rounded rectangle at (120,248)-(151,264): text "%.1f"; shows WORD_TO_REAL(CronEd.PR.Setpoint[123])/10; runs INTERN ASSIGN CronEd.PR.Setpoint[123]:=(REAL_TO_WORD(CronEd.PR_TT*10))
rounded rectangle at (120,262)-(151,278): text "%.1f"; shows WORD_TO_REAL(CronEd.PR.Setpoint[124])/10; runs INTERN ASSIGN CronEd.PR.Setpoint[124]:=(REAL_TO_WORD(CronEd.PR_TT*10))
rounded rectangle at (120,277)-(151,293): text "%.1f"; shows WORD_TO_REAL(CronEd.PR.Setpoint[125])/10; runs INTERN ASSIGN CronEd.PR.Setpoint[125]:=(REAL_TO_WORD(CronEd.PR_TT*10))
rounded rectangle at (120,292)-(151,308): text "%.1f"; shows WORD_TO_REAL(CronEd.PR.Setpoint[126])/10; runs INTERN ASSIGN CronEd.PR.Setpoint[126]:=(REAL_TO_WORD(CronEd.PR_TT*10))
rounded rectangle at (120,307)-(151,323): text "%.1f"; shows WORD_TO_REAL(CronEd.PR.Setpoint[127])/10; runs INTERN ASSIGN CronEd.PR.Setpoint[127]:=(REAL_TO_WORD(CronEd.PR_TT*10))
rounded rectangle at (120,321)-(151,337): text "%.1f"; shows WORD_TO_REAL(CronEd.PR.Setpoint[128])/10; runs INTERN ASSIGN CronEd.PR.Setpoint[128]:=(REAL_TO_WORD(CronEd.PR_TT*10))
rounded rectangle at (120,336)-(151,352): text "%.1f"; shows WORD_TO_REAL(CronEd.PR.Setpoint[129])/10; runs INTERN ASSIGN CronEd.PR.Setpoint[129]:=(REAL_TO_WORD(CronEd.PR_TT*10))
rounded rectangle at (120,351)-(151,367): text "%.1f"; shows WORD_TO_REAL(CronEd.PR.Setpoint[130])/10; runs INTERN ASSIGN CronEd.PR.Setpoint[130]:=(REAL_TO_WORD(CronEd.PR_TT*10))
rounded rectangle at (120,366)-(151,382): text "%.1f"; shows WORD_TO_REAL(CronEd.PR.Setpoint[131])/10; runs INTERN ASSIGN CronEd.PR.Setpoint[131]:=(REAL_TO_WORD(CronEd.PR_TT*10))
rounded rectangle at (120,380)-(151,396): text "%.1f"; shows WORD_TO_REAL(CronEd.PR.Setpoint[132])/10; runs INTERN ASSIGN CronEd.PR.Setpoint[132]:=(REAL_TO_WORD(CronEd.PR_TT*10))
rounded rectangle at (120,395)-(151,411): text "%.1f"; shows WORD_TO_REAL(CronEd.PR.Setpoint[133])/10; runs INTERN ASSIGN CronEd.PR.Setpoint[133]:=(REAL_TO_WORD(CronEd.PR_TT*10))
rounded rectangle at (120,410)-(151,426): text "%.1f"; shows WORD_TO_REAL(CronEd.PR.Setpoint[134])/10; runs INTERN ASSIGN CronEd.PR.Setpoint[134]:=(REAL_TO_WORD(CronEd.PR_TT*10))
rounded rectangle at (120,425)-(151,441): text "%.1f"; shows WORD_TO_REAL(CronEd.PR.Setpoint[135])/10; runs INTERN ASSIGN CronEd.PR.Setpoint[135]:=(REAL_TO_WORD(CronEd.PR_TT*10))
rounded rectangle at (120,440)-(151,456): text "%.1f"; shows WORD_TO_REAL(CronEd.PR.Setpoint[136])/10; runs INTERN ASSIGN CronEd.PR.Setpoint[136]:=(REAL_TO_WORD(CronEd.PR_TT*10))
rounded rectangle at (120,455)-(151,471): text "%.1f"; shows WORD_TO_REAL(CronEd.PR.Setpoint[137])/10; runs INTERN ASSIGN CronEd.PR.Setpoint[137]:=(REAL_TO_WORD(CronEd.PR_TT*10))
rounded rectangle at (120,470)-(151,486): text "%.1f"; shows WORD_TO_REAL(CronEd.PR.Setpoint[138])/10; runs INTERN ASSIGN CronEd.PR.Setpoint[138]:=(REAL_TO_WORD(CronEd.PR_TT*10))
rounded rectangle at (120,485)-(151,501): text "%.1f"; shows WORD_TO_REAL(CronEd.PR.Setpoint[139])/10; runs INTERN ASSIGN CronEd.PR.Setpoint[139]:=(REAL_TO_WORD(CronEd.PR_TT*10))
rounded rectangle at (120,499)-(151,515): text "%.1f"; shows WORD_TO_REAL(CronEd.PR.Setpoint[140])/10; runs INTERN ASSIGN CronEd.PR.Setpoint[140]:=(REAL_TO_WORD(CronEd.PR_TT*10))
rounded rectangle at (120,514)-(151,530): text "%.1f"; shows WORD_TO_REAL(CronEd.PR.Setpoint[141])/10; runs INTERN ASSIGN CronEd.PR.Setpoint[141]:=(REAL_TO_WORD(CronEd.PR_TT*10))
rounded rectangle at (120,529)-(151,545): text "%.1f"; shows WORD_TO_REAL(CronEd.PR.Setpoint[142])/10; runs INTERN ASSIGN CronEd.PR.Setpoint[142]:=(REAL_TO_WORD(CronEd.PR_TT*10))
rounded rectangle at (120,544)-(151,560): text "%.1f"; shows WORD_TO_REAL(CronEd.PR.Setpoint[143])/10; runs INTERN ASSIGN CronEd.PR.Setpoint[143]:=(REAL_TO_WORD(CronEd.PR_TT*10))
rounded rectangle at (120,558)-(151,574): text "%.1f"; shows WORD_TO_REAL(CronEd.PR.Setpoint[144])/10; runs INTERN ASSIGN CronEd.PR.Setpoint[144]:=(REAL_TO_WORD(CronEd.PR_TT*10))
rounded rectangle at (120,573)-(151,589): text "%.1f"; shows WORD_TO_REAL(CronEd.PR.Setpoint[145])/10; runs INTERN ASSIGN CronEd.PR.Setpoint[145]:=(REAL_TO_WORD(CronEd.PR_TT*10))
rounded rectangle at (120,588)-(151,604): text "%.1f"; shows WORD_TO_REAL(CronEd.PR.Setpoint[146])/10; runs INTERN ASSIGN CronEd.PR.Setpoint[146]:=(REAL_TO_WORD(CronEd.PR_TT*10))
rounded rectangle at (120,603)-(151,619): text "%.1f"; shows WORD_TO_REAL(CronEd.PR.Setpoint[147])/10; runs INTERN ASSIGN CronEd.PR.Setpoint[147]:=(REAL_TO_WORD(CronEd.PR_TT*10))
rounded rectangle at (120,617)-(151,633): text "%.1f"; shows WORD_TO_REAL(CronEd.PR.Setpoint[148])/10; runs INTERN ASSIGN CronEd.PR.Setpoint[148]:=(REAL_TO_WORD(CronEd.PR_TT*10))
rounded rectangle at (120,632)-(151,648): text "%.1f"; shows WORD_TO_REAL(CronEd.PR.Setpoint[149])/10; runs INTERN ASSIGN CronEd.PR.Setpoint[149]:=(REAL_TO_WORD(CronEd.PR_TT*10))
rounded rectangle at (120,647)-(151,663): text "%.1f"; shows WORD_TO_REAL(CronEd.PR.Setpoint[150])/10; runs INTERN ASSIGN CronEd.PR.Setpoint[150]:=(REAL_TO_WORD(CronEd.PR_TT*10))
rounded rectangle at (120,662)-(151,678): text "%.1f"; shows WORD_TO_REAL(CronEd.PR.Setpoint[151])/10; runs INTERN ASSIGN CronEd.PR.Setpoint[151]:=(REAL_TO_WORD(CronEd.PR_TT*10))
rounded rectangle at (570,677)-(601,693): text "%.1f"; shows WORD_TO_REAL(CronEd.PR.Setpoint[92])/10; runs INTERN ASSIGN CronEd.PR.Setpoint[92]:=(REAL_TO_WORD(CronEd.PR_TT*10))
rounded rectangle at (570,692)-(601,708): text "%.1f"; shows WORD_TO_REAL(CronEd.PR.Setpoint[93])/10; runs INTERN ASSIGN CronEd.PR.Setpoint[93]:=(REAL_TO_WORD(CronEd.PR_TT*10))
rounded rectangle at (570,707)-(601,723): text "%.1f"; shows WORD_TO_REAL(CronEd.PR.Setpoint[94])/10; runs INTERN ASSIGN CronEd.PR.Setpoint[94]:=(REAL_TO_WORD(CronEd.PR_TT*10))
rounded rectangle at (570,722)-(601,738): text "%.1f"; shows WORD_TO_REAL(CronEd.PR.Setpoint[95])/10; runs INTERN ASSIGN CronEd.PR.Setpoint[95]:=(REAL_TO_WORD(CronEd.PR_TT*10))
rounded rectangle at (570,737)-(601,753): text "%.1f"; shows WORD_TO_REAL(CronEd.PR.Setpoint[96])/10; runs INTERN ASSIGN CronEd.PR.Setpoint[96]:=(REAL_TO_WORD(CronEd.PR_TT*10))
rounded rectangle at (570,752)-(601,768): text "%.1f"; shows WORD_TO_REAL(CronEd.PR.Setpoint[97])/10; runs INTERN ASSIGN CronEd.PR.Setpoint[97]:=(REAL_TO_WORD(CronEd.PR_TT*10))
rounded rectangle at (570,767)-(601,783): text "%.1f"; shows WORD_TO_REAL(CronEd.PR.Setpoint[98])/10; runs INTERN ASSIGN CronEd.PR.Setpoint[98]:=(REAL_TO_WORD(CronEd.PR_TT*10))
rounded rectangle at (570,782)-(601,798): text "%.1f"; shows WORD_TO_REAL(CronEd.PR.Setpoint[99])/10; runs INTERN ASSIGN CronEd.PR.Setpoint[99]:=(REAL_TO_WORD(CronEd.PR_TT*10))
rounded rectangle at (570,796)-(601,812): text "%.1f"; shows WORD_TO_REAL(CronEd.PR.Setpoint[100])/10; runs INTERN ASSIGN CronEd.PR.Setpoint[100]:=(REAL_TO_WORD(CronEd.PR_TT*10))
rounded rectangle at (570,811)-(601,827): text "%.1f"; shows WORD_TO_REAL(CronEd.PR.Setpoint[101])/10; runs INTERN ASSIGN CronEd.PR.Setpoint[101]:=(REAL_TO_WORD(CronEd.PR_TT*10))
rounded rectangle at (570,826)-(601,842): text "%.1f"; shows WORD_TO_REAL(CronEd.PR.Setpoint[102])/10; runs INTERN ASSIGN CronEd.PR.Setpoint[102]:=(REAL_TO_WORD(CronEd.PR_TT*10))
rounded rectangle at (570,841)-(601,857): text "%.1f"; shows WORD_TO_REAL(CronEd.PR.Setpoint[103])/10; runs INTERN ASSIGN CronEd.PR.Setpoint[103]:=(REAL_TO_WORD(CronEd.PR_TT*10))
rounded rectangle at (570,855)-(601,871): text "%.1f"; shows WORD_TO_REAL(CronEd.PR.Setpoint[104])/10; runs INTERN ASSIGN CronEd.PR.Setpoint[104]:=(REAL_TO_WORD(CronEd.PR_TT*10))
rounded rectangle at (570,870)-(601,886): text "%.1f"; shows WORD_TO_REAL(CronEd.PR.Setpoint[105])/10; runs INTERN ASSIGN CronEd.PR.Setpoint[105]:=(REAL_TO_WORD(CronEd.PR_TT*10))
rounded rectangle at (570,885)-(601,901): text "%.1f"; shows WORD_TO_REAL(CronEd.PR.Setpoint[106])/10; runs INTERN ASSIGN CronEd.PR.Setpoint[106]:=(REAL_TO_WORD(CronEd.PR_TT*10))
rounded rectangle at (570,900)-(601,916): text "%.1f"; shows WORD_TO_REAL(CronEd.PR.Setpoint[107])/10; runs INTERN ASSIGN CronEd.PR.Setpoint[107]:=(REAL_TO_WORD(CronEd.PR_TT*10))
rounded rectangle at (570,914)-(601,930): text "%.1f"; shows WORD_TO_REAL(CronEd.PR.Setpoint[1068])/10; runs INTERN ASSIGN CronEd.PR.Setpoint[1068]:=(REAL_TO_WORD(CronEd.PR_TT*10))
rounded rectangle at (570,929)-(601,945): text "%.1f"; shows WORD_TO_REAL(CronEd.PR.Setpoint[1069])/10; runs INTERN ASSIGN CronEd.PR.Setpoint[1069]:=(REAL_TO_WORD(CronEd.PR_TT*10))
rounded rectangle at (570,944)-(601,960): text "%.1f"; shows WORD_TO_REAL(CronEd.PR.Setpoint[1070])/10; runs INTERN ASSIGN CronEd.PR.Setpoint[1070]:=(REAL_TO_WORD(CronEd.PR_TT*10))
rounded rectangle at (570,959)-(601,975): text "%.1f"; shows WORD_TO_REAL(CronEd.PR.Setpoint[1071])/10; runs INTERN ASSIGN CronEd.PR.Setpoint[1071]:=(REAL_TO_WORD(CronEd.PR_TT*10))
rounded rectangle at (570,973)-(601,989): text "%.1f"; shows WORD_TO_REAL(CronEd.PR.Setpoint[1072])/10; runs INTERN ASSIGN CronEd.PR.Setpoint[1072]:=(REAL_TO_WORD(CronEd.PR_TT*10))
rounded rectangle at (570,988)-(601,1004): text "%.1f"; shows WORD_TO_REAL(CronEd.PR.Setpoint[1073])/10; runs INTERN ASSIGN CronEd.PR.Setpoint[1073]:=(REAL_TO_WORD(CronEd.PR_TT*10))
rounded rectangle at (570,1003)-(601,1019): text "%.1f"; shows WORD_TO_REAL(CronEd.PR.Setpoint[1074])/10; runs INTERN ASSIGN CronEd.PR.Setpoint[1074]:=(REAL_TO_WORD(CronEd.PR_TT*10))
rounded rectangle at (570,1018)-(601,1034): text "%.1f"; shows WORD_TO_REAL(CronEd.PR.Setpoint[1075])/10; runs INTERN ASSIGN CronEd.PR.Setpoint[1075]:=(REAL_TO_WORD(CronEd.PR_TT*10))
rounded rectangle at (570,1033)-(601,1049): text "%.1f"; shows WORD_TO_REAL(CronEd.PR.Setpoint[1076])/10; runs INTERN ASSIGN CronEd.PR.Setpoint[1076]:=(REAL_TO_WORD(CronEd.PR_TT*10))
rounded rectangle at (570,1048)-(601,1064): text "%.1f"; shows WORD_TO_REAL(CronEd.PR.Setpoint[1077])/10; runs INTERN ASSIGN CronEd.PR.Setpoint[1077]:=(REAL_TO_WORD(CronEd.PR_TT*10))
rounded rectangle at (570,1063)-(601,1079): text "%.1f"; shows WORD_TO_REAL(CronEd.PR.Setpoint[1078])/10; runs INTERN ASSIGN CronEd.PR.Setpoint[1078]:=(REAL_TO_WORD(CronEd.PR_TT*10))
rounded rectangle at (570,1078)-(601,1094): text "%.1f"; shows WORD_TO_REAL(CronEd.PR.Setpoint[1079])/10; runs INTERN ASSIGN CronEd.PR.Setpoint[1079]:=(REAL_TO_WORD(CronEd.PR_TT*10))
group at (90,203)-(121,1093)
  rounded rectangle at (0,0)-(31,16): text "%.1f"; shows WORD_TO_REAL(CronEd.PR.Setpoint[60])/10; runs INTERN ASSIGN CronEd.PR.Setpoint[60]:=(REAL_TO_WORD(CronEd.PR_TT*10))
  rounded rectangle at (0,15)-(31,31): text "%.1f"; shows WORD_TO_REAL(CronEd.PR.Setpoint[61])/10; runs INTERN ASSIGN CronEd.PR.Setpoint[61]:=(REAL_TO_WORD(CronEd.PR_TT*10))
  rounded rectangle at (0,30)-(31,46): text "%.1f"; shows WORD_TO_REAL(CronEd.PR.Setpoint[62])/10; runs INTERN ASSIGN CronEd.PR.Setpoint[62]:=(REAL_TO_WORD(CronEd.PR_TT*10))
  rounded rectangle at (0,45)-(31,61): text "%.1f"; shows WORD_TO_REAL(CronEd.PR.Setpoint[63])/10; runs INTERN ASSIGN CronEd.PR.Setpoint[63]:=(REAL_TO_WORD(CronEd.PR_TT*10))
  rounded rectangle at (0,59)-(31,75): text "%.1f"; shows WORD_TO_REAL(CronEd.PR.Setpoint[64])/10; runs INTERN ASSIGN CronEd.PR.Setpoint[64]:=(REAL_TO_WORD(CronEd.PR_TT*10))
  rounded rectangle at (0,74)-(31,90): text "%.1f"; shows WORD_TO_REAL(CronEd.PR.Setpoint[65])/10; runs INTERN ASSIGN CronEd.PR.Setpoint[65]:=(REAL_TO_WORD(CronEd.PR_TT*10))
  rounded rectangle at (0,89)-(31,105): text "%.1f"; shows WORD_TO_REAL(CronEd.PR.Setpoint[66])/10; runs INTERN ASSIGN CronEd.PR.Setpoint[66]:=(REAL_TO_WORD(CronEd.PR_TT*10))
  rounded rectangle at (0,104)-(31,120): text "%.1f"; shows WORD_TO_REAL(CronEd.PR.Setpoint[67])/10; runs INTERN ASSIGN CronEd.PR.Setpoint[67]:=(REAL_TO_WORD(CronEd.PR_TT*10))
  rounded rectangle at (0,118)-(31,134): text "%.1f"; shows WORD_TO_REAL(CronEd.PR.Setpoint[68])/10; runs INTERN ASSIGN CronEd.PR.Setpoint[68]:=(REAL_TO_WORD(CronEd.PR_TT*10))
  rounded rectangle at (0,133)-(31,149): text "%.1f"; shows WORD_TO_REAL(CronEd.PR.Setpoint[69])/10; runs INTERN ASSIGN CronEd.PR.Setpoint[69]:=(REAL_TO_WORD(CronEd.PR_TT*10))
  rounded rectangle at (0,148)-(31,164): text "%.1f"; shows WORD_TO_REAL(CronEd.PR.Setpoint[70])/10; runs INTERN ASSIGN CronEd.PR.Setpoint[70]:=(REAL_TO_WORD(CronEd.PR_TT*10))
  rounded rectangle at (0,163)-(31,179): text "%.1f"; shows WORD_TO_REAL(CronEd.PR.Setpoint[71])/10; runs INTERN ASSIGN CronEd.PR.Setpoint[71]:=(REAL_TO_WORD(CronEd.PR_TT*10))
  rounded rectangle at (0,177)-(31,193): text "%.1f"; shows WORD_TO_REAL(CronEd.PR.Setpoint[72])/10; runs INTERN ASSIGN CronEd.PR.Setpoint[72]:=(REAL_TO_WORD(CronEd.PR_TT*10))
  rounded rectangle at (0,192)-(31,208): text "%.1f"; shows WORD_TO_REAL(CronEd.PR.Setpoint[73])/10; runs INTERN ASSIGN CronEd.PR.Setpoint[73]:=(REAL_TO_WORD(CronEd.PR_TT*10))
  rounded rectangle at (0,207)-(31,223): text "%.1f"; shows WORD_TO_REAL(CronEd.PR.Setpoint[74])/10; runs INTERN ASSIGN CronEd.PR.Setpoint[74]:=(REAL_TO_WORD(CronEd.PR_TT*10))
  rounded rectangle at (0,222)-(31,238): text "%.1f"; shows WORD_TO_REAL(CronEd.PR.Setpoint[75])/10; runs INTERN ASSIGN CronEd.PR.Setpoint[75]:=(REAL_TO_WORD(CronEd.PR_TT*10))
  rounded rectangle at (0,237)-(31,253): text "%.1f"; shows WORD_TO_REAL(CronEd.PR.Setpoint[76])/10; runs INTERN ASSIGN CronEd.PR.Setpoint[76]:=(REAL_TO_WORD(CronEd.PR_TT*10))
  rounded rectangle at (0,252)-(31,268): text "%.1f"; shows WORD_TO_REAL(CronEd.PR.Setpoint[77])/10; runs INTERN ASSIGN CronEd.PR.Setpoint[77]:=(REAL_TO_WORD(CronEd.PR_TT*10))
  rounded rectangle at (0,267)-(31,283): text "%.1f"; shows WORD_TO_REAL(CronEd.PR.Setpoint[78])/10; runs INTERN ASSIGN CronEd.PR.Setpoint[78]:=(REAL_TO_WORD(CronEd.PR_TT*10))
  rounded rectangle at (0,282)-(31,298): text "%.1f"; shows WORD_TO_REAL(CronEd.PR.Setpoint[79])/10; runs INTERN ASSIGN CronEd.PR.Setpoint[79]:=(REAL_TO_WORD(CronEd.PR_TT*10))
  rounded rectangle at (0,296)-(31,312): text "%.1f"; shows WORD_TO_REAL(CronEd.PR.Setpoint[80])/10; runs INTERN ASSIGN CronEd.PR.Setpoint[80]:=(REAL_TO_WORD(CronEd.PR_TT*10))
  rounded rectangle at (0,311)-(31,327): text "%.1f"; shows WORD_TO_REAL(CronEd.PR.Setpoint[81])/10; runs INTERN ASSIGN CronEd.PR.Setpoint[81]:=(REAL_TO_WORD(CronEd.PR_TT*10))
  rounded rectangle at (0,326)-(31,342): text "%.1f"; shows WORD_TO_REAL(CronEd.PR.Setpoint[82])/10; runs INTERN ASSIGN CronEd.PR.Setpoint[82]:=(REAL_TO_WORD(CronEd.PR_TT*10))
  rounded rectangle at (0,341)-(31,357): text "%.1f"; shows WORD_TO_REAL(CronEd.PR.Setpoint[83])/10; runs INTERN ASSIGN CronEd.PR.Setpoint[83]:=(REAL_TO_WORD(CronEd.PR_TT*10))
  rounded rectangle at (0,355)-(31,371): text "%.1f"; shows WORD_TO_REAL(CronEd.PR.Setpoint[84])/10; runs INTERN ASSIGN CronEd.PR.Setpoint[84]:=(REAL_TO_WORD(CronEd.PR_TT*10))
  rounded rectangle at (0,370)-(31,386): text "%.1f"; shows WORD_TO_REAL(CronEd.PR.Setpoint[85])/10; runs INTERN ASSIGN CronEd.PR.Setpoint[85]:=(REAL_TO_WORD(CronEd.PR_TT*10))
  rounded rectangle at (0,385)-(31,401): text "%.1f"; shows WORD_TO_REAL(CronEd.PR.Setpoint[86])/10; runs INTERN ASSIGN CronEd.PR.Setpoint[86]:=(REAL_TO_WORD(CronEd.PR_TT*10))
  rounded rectangle at (0,400)-(31,416): text "%.1f"; shows WORD_TO_REAL(CronEd.PR.Setpoint[87])/10; runs INTERN ASSIGN CronEd.PR.Setpoint[87]:=(REAL_TO_WORD(CronEd.PR_TT*10))
  rounded rectangle at (0,414)-(31,430): text "%.1f"; shows WORD_TO_REAL(CronEd.PR.Setpoint[88])/10; runs INTERN ASSIGN CronEd.PR.Setpoint[88]:=(REAL_TO_WORD(CronEd.PR_TT*10))
  rounded rectangle at (0,429)-(31,445): text "%.1f"; shows WORD_TO_REAL(CronEd.PR.Setpoint[89])/10; runs INTERN ASSIGN CronEd.PR.Setpoint[89]:=(REAL_TO_WORD(CronEd.PR_TT*10))
  rounded rectangle at (0,444)-(31,460): text "%.1f"; shows WORD_TO_REAL(CronEd.PR.Setpoint[90])/10; runs INTERN ASSIGN CronEd.PR.Setpoint[90]:=(REAL_TO_WORD(CronEd.PR_TT*10))
  rounded rectangle at (0,459)-(31,475): text "%.1f"; shows WORD_TO_REAL(CronEd.PR.Setpoint[91])/10; runs INTERN ASSIGN CronEd.PR.Setpoint[91]:=(REAL_TO_WORD(CronEd.PR_TT*10))
  rounded rectangle at (0,473)-(31,489): text "%.1f"; shows WORD_TO_REAL(CronEd.PR.Setpoint[92])/10; runs INTERN ASSIGN CronEd.PR.Setpoint[92]:=(REAL_TO_WORD(CronEd.PR_TT*10))
  rounded rectangle at (0,488)-(31,504): text "%.1f"; shows WORD_TO_REAL(CronEd.PR.Setpoint[93])/10; runs INTERN ASSIGN CronEd.PR.Setpoint[93]:=(REAL_TO_WORD(CronEd.PR_TT*10))
  rounded rectangle at (0,503)-(31,519): text "%.1f"; shows WORD_TO_REAL(CronEd.PR.Setpoint[94])/10; runs INTERN ASSIGN CronEd.PR.Setpoint[94]:=(REAL_TO_WORD(CronEd.PR_TT*10))
  rounded rectangle at (0,518)-(31,534): text "%.1f"; shows WORD_TO_REAL(CronEd.PR.Setpoint[95])/10; runs INTERN ASSIGN CronEd.PR.Setpoint[95]:=(REAL_TO_WORD(CronEd.PR_TT*10))
  rounded rectangle at (0,533)-(31,549): text "%.1f"; shows WORD_TO_REAL(CronEd.PR.Setpoint[96])/10; runs INTERN ASSIGN CronEd.PR.Setpoint[96]:=(REAL_TO_WORD(CronEd.PR_TT*10))
  rounded rectangle at (0,548)-(31,564): text "%.1f"; shows WORD_TO_REAL(CronEd.PR.Setpoint[97])/10; runs INTERN ASSIGN CronEd.PR.Setpoint[97]:=(REAL_TO_WORD(CronEd.PR_TT*10))
  rounded rectangle at (0,563)-(31,579): text "%.1f"; shows WORD_TO_REAL(CronEd.PR.Setpoint[98])/10; runs INTERN ASSIGN CronEd.PR.Setpoint[98]:=(REAL_TO_WORD(CronEd.PR_TT*10))
  rounded rectangle at (0,578)-(31,594): text "%.1f"; shows WORD_TO_REAL(CronEd.PR.Setpoint[99])/10; runs INTERN ASSIGN CronEd.PR.Setpoint[99]:=(REAL_TO_WORD(CronEd.PR_TT*10))
  rounded rectangle at (0,592)-(31,608): text "%.1f"; shows WORD_TO_REAL(CronEd.PR.Setpoint[100])/10; runs INTERN ASSIGN CronEd.PR.Setpoint[100]:=(REAL_TO_WORD(CronEd.PR_TT*10))
  rounded rectangle at (0,607)-(31,623): text "%.1f"; shows WORD_TO_REAL(CronEd.PR.Setpoint[101])/10; runs INTERN ASSIGN CronEd.PR.Setpoint[101]:=(REAL_TO_WORD(CronEd.PR_TT*10))
  rounded rectangle at (0,622)-(31,638): text "%.1f"; shows WORD_TO_REAL(CronEd.PR.Setpoint[102])/10; runs INTERN ASSIGN CronEd.PR.Setpoint[102]:=(REAL_TO_WORD(CronEd.PR_TT*10))
  rounded rectangle at (0,637)-(31,653): text "%.1f"; shows WORD_TO_REAL(CronEd.PR.Setpoint[103])/10; runs INTERN ASSIGN CronEd.PR.Setpoint[103]:=(REAL_TO_WORD(CronEd.PR_TT*10))
  rounded rectangle at (0,651)-(31,667): text "%.1f"; shows WORD_TO_REAL(CronEd.PR.Setpoint[104])/10; runs INTERN ASSIGN CronEd.PR.Setpoint[104]:=(REAL_TO_WORD(CronEd.PR_TT*10))
  rounded rectangle at (0,666)-(31,682): text "%.1f"; shows WORD_TO_REAL(CronEd.PR.Setpoint[105])/10; runs INTERN ASSIGN CronEd.PR.Setpoint[105]:=(REAL_TO_WORD(CronEd.PR_TT*10))
  rounded rectangle at (0,681)-(31,697): text "%.1f"; shows WORD_TO_REAL(CronEd.PR.Setpoint[106])/10; runs INTERN ASSIGN CronEd.PR.Setpoint[106]:=(REAL_TO_WORD(CronEd.PR_TT*10))
  rounded rectangle at (0,696)-(31,712): text "%.1f"; shows WORD_TO_REAL(CronEd.PR.Setpoint[107])/10; runs INTERN ASSIGN CronEd.PR.Setpoint[107]:=(REAL_TO_WORD(CronEd.PR_TT*10))
  rounded rectangle at (0,710)-(31,726): text "%.1f"; shows WORD_TO_REAL(CronEd.PR.Setpoint[108])/10; runs INTERN ASSIGN CronEd.PR.Setpoint[108]:=(REAL_TO_WORD(CronEd.PR_TT*10))
  rounded rectangle at (0,725)-(31,741): text "%.1f"; shows WORD_TO_REAL(CronEd.PR.Setpoint[109])/10; runs INTERN ASSIGN CronEd.PR.Setpoint[109]:=(REAL_TO_WORD(CronEd.PR_TT*10))
  rounded rectangle at (0,740)-(31,756): text "%.1f"; shows WORD_TO_REAL(CronEd.PR.Setpoint[110])/10; runs INTERN ASSIGN CronEd.PR.Setpoint[110]:=(REAL_TO_WORD(CronEd.PR_TT*10))
  rounded rectangle at (0,755)-(31,771): text "%.1f"; shows WORD_TO_REAL(CronEd.PR.Setpoint[111])/10; runs INTERN ASSIGN CronEd.PR.Setpoint[111]:=(REAL_TO_WORD(CronEd.PR_TT*10))
  rounded rectangle at (0,769)-(31,785): text "%.1f"; shows WORD_TO_REAL(CronEd.PR.Setpoint[112])/10; runs INTERN ASSIGN CronEd.PR.Setpoint[112]:=(REAL_TO_WORD(CronEd.PR_TT*10))
  rounded rectangle at (0,784)-(31,800): text "%.1f"; shows WORD_TO_REAL(CronEd.PR.Setpoint[113])/10; runs INTERN ASSIGN CronEd.PR.Setpoint[113]:=(REAL_TO_WORD(CronEd.PR_TT*10))
  rounded rectangle at (0,799)-(31,815): text "%.1f"; shows WORD_TO_REAL(CronEd.PR.Setpoint[114])/10; runs INTERN ASSIGN CronEd.PR.Setpoint[114]:=(REAL_TO_WORD(CronEd.PR_TT*10))
  rounded rectangle at (0,814)-(31,830): text "%.1f"; shows WORD_TO_REAL(CronEd.PR.Setpoint[115])/10; runs INTERN ASSIGN CronEd.PR.Setpoint[115]:=(REAL_TO_WORD(CronEd.PR_TT*10))
  rounded rectangle at (0,829)-(31,845): text "%.1f"; shows WORD_TO_REAL(CronEd.PR.Setpoint[116])/10; runs INTERN ASSIGN CronEd.PR.Setpoint[116]:=(REAL_TO_WORD(CronEd.PR_TT*10))
  rounded rectangle at (0,844)-(31,860): text "%.1f"; shows WORD_TO_REAL(CronEd.PR.Setpoint[117])/10; runs INTERN ASSIGN CronEd.PR.Setpoint[117]:=(REAL_TO_WORD(CronEd.PR_TT*10))
  rounded rectangle at (0,859)-(31,875): text "%.1f"; shows WORD_TO_REAL(CronEd.PR.Setpoint[118])/10; runs INTERN ASSIGN CronEd.PR.Setpoint[118]:=(REAL_TO_WORD(CronEd.PR_TT*10))
  rounded rectangle at (0,874)-(31,890): text "%.1f"; shows WORD_TO_REAL(CronEd.PR.Setpoint[119])/10; runs INTERN ASSIGN CronEd.PR.Setpoint[119]:=(REAL_TO_WORD(CronEd.PR_TT*10))
rounded rectangle at (60,203)-(91,219): text "%.1f"; shows WORD_TO_REAL(CronEd.PR.Setpoint[0])/10; runs INTERN ASSIGN CronEd.PR.Setpoint[0]:=(REAL_TO_WORD(CronEd.PR_TT*10))
rounded rectangle at (60,218)-(91,234): text "%.1f"; shows WORD_TO_REAL(CronEd.PR.Setpoint[1])/10; runs INTERN ASSIGN CronEd.PR.Setpoint[1]:=(REAL_TO_WORD(CronEd.PR_TT*10))
rounded rectangle at (60,233)-(91,249): text "%.1f"; shows WORD_TO_REAL(CronEd.PR.Setpoint[2])/10; runs INTERN ASSIGN CronEd.PR.Setpoint[2]:=(REAL_TO_WORD(CronEd.PR_TT*10))
rounded rectangle at (60,248)-(91,264): text "%.1f"; shows WORD_TO_REAL(CronEd.PR.Setpoint[3])/10; runs INTERN ASSIGN CronEd.PR.Setpoint[3]:=(REAL_TO_WORD(CronEd.PR_TT*10))
rounded rectangle at (60,262)-(91,278): text "%.1f"; shows WORD_TO_REAL(CronEd.PR.Setpoint[4])/10; runs INTERN ASSIGN CronEd.PR.Setpoint[4]:=(REAL_TO_WORD(CronEd.PR_TT*10))
rounded rectangle at (60,277)-(91,293): text "%.1f"; shows WORD_TO_REAL(CronEd.PR.Setpoint[5])/10; runs INTERN ASSIGN CronEd.PR.Setpoint[5]:=(REAL_TO_WORD(CronEd.PR_TT*10))
rounded rectangle at (60,292)-(91,308): text "%.1f"; shows WORD_TO_REAL(CronEd.PR.Setpoint[6])/10; runs INTERN ASSIGN CronEd.PR.Setpoint[6]:=(REAL_TO_WORD(CronEd.PR_TT*10))
rounded rectangle at (60,307)-(91,323): text "%.1f"; shows WORD_TO_REAL(CronEd.PR.Setpoint[7])/10; runs INTERN ASSIGN CronEd.PR.Setpoint[7]:=(REAL_TO_WORD(CronEd.PR_TT*10))
rounded rectangle at (60,321)-(91,337): text "%.1f"; shows WORD_TO_REAL(CronEd.PR.Setpoint[8])/10; runs INTERN ASSIGN CronEd.PR.Setpoint[8]:=(REAL_TO_WORD(CronEd.PR_TT*10))
rounded rectangle at (60,336)-(91,352): text "%.1f"; shows WORD_TO_REAL(CronEd.PR.Setpoint[9])/10; runs INTERN ASSIGN CronEd.PR.Setpoint[9]:=(REAL_TO_WORD(CronEd.PR_TT*10))
rounded rectangle at (60,351)-(91,367): text "%.1f"; shows WORD_TO_REAL(CronEd.PR.Setpoint[10])/10; runs INTERN ASSIGN CronEd.PR.Setpoint[10]:=(REAL_TO_WORD(CronEd.PR_TT*10))
rounded rectangle at (60,366)-(91,382): text "%.1f"; shows WORD_TO_REAL(CronEd.PR.Setpoint[11])/10; runs INTERN ASSIGN CronEd.PR.Setpoint[11]:=(REAL_TO_WORD(CronEd.PR_TT*10))
rounded rectangle at (60,381)-(91,397): text "%.1f"; shows WORD_TO_REAL(CronEd.PR.Setpoint[12])/10; runs INTERN ASSIGN CronEd.PR.Setpoint[12]:=(REAL_TO_WORD(CronEd.PR_TT*10))
rounded rectangle at (60,396)-(91,412): text "%.1f"; shows WORD_TO_REAL(CronEd.PR.Setpoint[13])/10; runs INTERN ASSIGN CronEd.PR.Setpoint[13]:=(REAL_TO_WORD(CronEd.PR_TT*10))
rounded rectangle at (60,411)-(91,427): text "%.1f"; shows WORD_TO_REAL(CronEd.PR.Setpoint[14])/10; runs INTERN ASSIGN CronEd.PR.Setpoint[14]:=(REAL_TO_WORD(CronEd.PR_TT*10))
rounded rectangle at (60,426)-(91,442): text "%.1f"; shows WORD_TO_REAL(CronEd.PR.Setpoint[15])/10; runs INTERN ASSIGN CronEd.PR.Setpoint[15]:=(REAL_TO_WORD(CronEd.PR_TT*10))
rounded rectangle at (60,441)-(91,457): text "%.1f"; shows WORD_TO_REAL(CronEd.PR.Setpoint[16])/10; runs INTERN ASSIGN CronEd.PR.Setpoint[16]:=(REAL_TO_WORD(CronEd.PR_TT*10))
rounded rectangle at (60,456)-(91,472): text "%.1f"; shows WORD_TO_REAL(CronEd.PR.Setpoint[17])/10; runs INTERN ASSIGN CronEd.PR.Setpoint[17]:=(REAL_TO_WORD(CronEd.PR_TT*10))
rounded rectangle at (60,471)-(91,487): text "%.1f"; shows WORD_TO_REAL(CronEd.PR.Setpoint[18])/10; runs INTERN ASSIGN CronEd.PR.Setpoint[18]:=(REAL_TO_WORD(CronEd.PR_TT*10))
rounded rectangle at (60,486)-(91,502): text "%.1f"; shows WORD_TO_REAL(CronEd.PR.Setpoint[19])/10; runs INTERN ASSIGN CronEd.PR.Setpoint[19]:=(REAL_TO_WORD(CronEd.PR_TT*10))
rounded rectangle at (60,500)-(91,516): text "%.1f"; shows WORD_TO_REAL(CronEd.PR.Setpoint[20])/10; runs INTERN ASSIGN CronEd.PR.Setpoint[20]:=(REAL_TO_WORD(CronEd.PR_TT*10))
rounded rectangle at (60,515)-(91,531): text "%.1f"; shows WORD_TO_REAL(CronEd.PR.Setpoint[21])/10; runs INTERN ASSIGN CronEd.PR.Setpoint[21]:=(REAL_TO_WORD(CronEd.PR_TT*10))
rounded rectangle at (60,530)-(91,546): text "%.1f"; shows WORD_TO_REAL(CronEd.PR.Setpoint[22])/10; runs INTERN ASSIGN CronEd.PR.Setpoint[22]:=(REAL_TO_WORD(CronEd.PR_TT*10))
rounded rectangle at (60,545)-(91,561): text "%.1f"; shows WORD_TO_REAL(CronEd.PR.Setpoint[23])/10; runs INTERN ASSIGN CronEd.PR.Setpoint[23]:=(REAL_TO_WORD(CronEd.PR_TT*10))
rounded rectangle at (60,559)-(91,575): text "%.1f"; shows WORD_TO_REAL(CronEd.PR.Setpoint[24])/10; runs INTERN ASSIGN CronEd.PR.Setpoint[24]:=(REAL_TO_WORD(CronEd.PR_TT*10))
rounded rectangle at (60,574)-(91,590): text "%.1f"; shows WORD_TO_REAL(CronEd.PR.Setpoint[25])/10; runs INTERN ASSIGN CronEd.PR.Setpoint[25]:=(REAL_TO_WORD(CronEd.PR_TT*10))
rounded rectangle at (60,589)-(91,605): text "%.1f"; shows WORD_TO_REAL(CronEd.PR.Setpoint[26])/10; runs INTERN ASSIGN CronEd.PR.Setpoint[26]:=(REAL_TO_WORD(CronEd.PR_TT*10))
rounded rectangle at (60,604)-(91,620): text "%.1f"; shows WORD_TO_REAL(CronEd.PR.Setpoint[27])/10; runs INTERN ASSIGN CronEd.PR.Setpoint[27]:=(REAL_TO_WORD(CronEd.PR_TT*10))
rounded rectangle at (60,618)-(91,634): text "%.1f"; shows WORD_TO_REAL(CronEd.PR.Setpoint[28])/10; runs INTERN ASSIGN CronEd.PR.Setpoint[28]:=(REAL_TO_WORD(CronEd.PR_TT*10))
rounded rectangle at (60,633)-(91,649): text "%.1f"; shows WORD_TO_REAL(CronEd.PR.Setpoint[29])/10; runs INTERN ASSIGN CronEd.PR.Setpoint[29]:=(REAL_TO_WORD(CronEd.PR_TT*10))
rounded rectangle at (60,648)-(91,664): text "%.1f"; shows WORD_TO_REAL(CronEd.PR.Setpoint[30])/10; runs INTERN ASSIGN CronEd.PR.Setpoint[30]:=(REAL_TO_WORD(CronEd.PR_TT*10))
rounded rectangle at (60,663)-(91,679): text "%.1f"; shows WORD_TO_REAL(CronEd.PR.Setpoint[31])/10; runs INTERN ASSIGN CronEd.PR.Setpoint[31]:=(REAL_TO_WORD(CronEd.PR_TT*10))
rounded rectangle at (60,677)-(91,693): text "%.1f"; shows WORD_TO_REAL(CronEd.PR.Setpoint[32])/10; runs INTERN ASSIGN CronEd.PR.Setpoint[32]:=(REAL_TO_WORD(CronEd.PR_TT*10))
rounded rectangle at (60,692)-(91,708): text "%.1f"; shows WORD_TO_REAL(CronEd.PR.Setpoint[33])/10; runs INTERN ASSIGN CronEd.PR.Setpoint[33]:=(REAL_TO_WORD(CronEd.PR_TT*10))
rounded rectangle at (60,707)-(91,723): text "%.1f"; shows WORD_TO_REAL(CronEd.PR.Setpoint[34])/10; runs INTERN ASSIGN CronEd.PR.Setpoint[34]:=(REAL_TO_WORD(CronEd.PR_TT*10))
rounded rectangle at (60,722)-(91,738): text "%.1f"; shows WORD_TO_REAL(CronEd.PR.Setpoint[35])/10; runs INTERN ASSIGN CronEd.PR.Setpoint[35]:=(REAL_TO_WORD(CronEd.PR_TT*10))
rounded rectangle at (60,737)-(91,753): text "%.1f"; shows WORD_TO_REAL(CronEd.PR.Setpoint[36])/10; runs INTERN ASSIGN CronEd.PR.Setpoint[36]:=(REAL_TO_WORD(CronEd.PR_TT*10))
rounded rectangle at (60,752)-(91,768): text "%.1f"; shows WORD_TO_REAL(CronEd.PR.Setpoint[37])/10; runs INTERN ASSIGN CronEd.PR.Setpoint[37]:=(REAL_TO_WORD(CronEd.PR_TT*10))
rounded rectangle at (60,767)-(91,783): text "%.1f"; shows WORD_TO_REAL(CronEd.PR.Setpoint[38])/10; runs INTERN ASSIGN CronEd.PR.Setpoint[38]:=(REAL_TO_WORD(CronEd.PR_TT*10))
rounded rectangle at (60,782)-(91,798): text "%.1f"; shows WORD_TO_REAL(CronEd.PR.Setpoint[39])/10; runs INTERN ASSIGN CronEd.PR.Setpoint[39]:=(REAL_TO_WORD(CronEd.PR_TT*10))
rounded rectangle at (60,796)-(91,812): text "%.1f"; shows WORD_TO_REAL(CronEd.PR.Setpoint[40])/10; runs INTERN ASSIGN CronEd.PR.Setpoint[40]:=(REAL_TO_WORD(CronEd.PR_TT*10))
rounded rectangle at (60,811)-(91,827): text "%.1f"; shows WORD_TO_REAL(CronEd.PR.Setpoint[41])/10; runs INTERN ASSIGN CronEd.PR.Setpoint[41]:=(REAL_TO_WORD(CronEd.PR_TT*10))
rounded rectangle at (60,826)-(91,842): text "%.1f"; shows WORD_TO_REAL(CronEd.PR.Setpoint[42])/10; runs INTERN ASSIGN CronEd.PR.Setpoint[42]:=(REAL_TO_WORD(CronEd.PR_TT*10))
rounded rectangle at (60,841)-(91,857): text "%.1f"; shows WORD_TO_REAL(CronEd.PR.Setpoint[43])/10; runs INTERN ASSIGN CronEd.PR.Setpoint[43]:=(REAL_TO_WORD(CronEd.PR_TT*10))
rounded rectangle at (60,855)-(91,871): text "%.1f"; shows WORD_TO_REAL(CronEd.PR.Setpoint[44])/10; runs INTERN ASSIGN CronEd.PR.Setpoint[44]:=(REAL_TO_WORD(CronEd.PR_TT*10))
rounded rectangle at (60,870)-(91,886): text "%.1f"; shows WORD_TO_REAL(CronEd.PR.Setpoint[45])/10; runs INTERN ASSIGN CronEd.PR.Setpoint[45]:=(REAL_TO_WORD(CronEd.PR_TT*10))
rounded rectangle at (60,885)-(91,901): text "%.1f"; shows WORD_TO_REAL(CronEd.PR.Setpoint[46])/10; runs INTERN ASSIGN CronEd.PR.Setpoint[46]:=(REAL_TO_WORD(CronEd.PR_TT*10))
rounded rectangle at (60,900)-(91,916): text "%.1f"; shows WORD_TO_REAL(CronEd.PR.Setpoint[47])/10; runs INTERN ASSIGN CronEd.PR.Setpoint[47]:=(REAL_TO_WORD(CronEd.PR_TT*10))
rounded rectangle at (59,914)-(90,930): text "%.1f"; shows WORD_TO_REAL(CronEd.PR.Setpoint[48])/10; runs INTERN ASSIGN CronEd.PR.Setpoint[48]:=(REAL_TO_WORD(CronEd.PR_TT*10))
rounded rectangle at (59,929)-(90,945): text "%.1f"; shows WORD_TO_REAL(CronEd.PR.Setpoint[49])/10; runs INTERN ASSIGN CronEd.PR.Setpoint[49]:=(REAL_TO_WORD(CronEd.PR_TT*10))
rounded rectangle at (59,944)-(90,960): text "%.1f"; shows WORD_TO_REAL(CronEd.PR.Setpoint[50])/10; runs INTERN ASSIGN CronEd.PR.Setpoint[50]:=(REAL_TO_WORD(CronEd.PR_TT*10))
rounded rectangle at (59,959)-(90,975): text "%.1f"; shows WORD_TO_REAL(CronEd.PR.Setpoint[51])/10; runs INTERN ASSIGN CronEd.PR.Setpoint[51]:=(REAL_TO_WORD(CronEd.PR_TT*10))
rounded rectangle at (58,973)-(89,989): text "%.1f"; shows WORD_TO_REAL(CronEd.PR.Setpoint[52])/10; runs INTERN ASSIGN CronEd.PR.Setpoint[52]:=(REAL_TO_WORD(CronEd.PR_TT*10))
rounded rectangle at (58,988)-(89,1004): text "%.1f"; shows WORD_TO_REAL(CronEd.PR.Setpoint[53])/10; runs INTERN ASSIGN CronEd.PR.Setpoint[53]:=(REAL_TO_WORD(CronEd.PR_TT*10))
rounded rectangle at (58,1003)-(89,1019): text "%.1f"; shows WORD_TO_REAL(CronEd.PR.Setpoint[54])/10; runs INTERN ASSIGN CronEd.PR.Setpoint[54]:=(REAL_TO_WORD(CronEd.PR_TT*10))
rounded rectangle at (58,1018)-(89,1034): text "%.1f"; shows WORD_TO_REAL(CronEd.PR.Setpoint[55])/10; runs INTERN ASSIGN CronEd.PR.Setpoint[55]:=(REAL_TO_WORD(CronEd.PR_TT*10))
rounded rectangle at (57,1033)-(88,1049): text "%.1f"; shows WORD_TO_REAL(CronEd.PR.Setpoint[56])/10; runs INTERN ASSIGN CronEd.PR.Setpoint[56]:=(REAL_TO_WORD(CronEd.PR_TT*10))
rounded rectangle at (57,1048)-(88,1064): text "%.1f"; shows WORD_TO_REAL(CronEd.PR.Setpoint[57])/10; runs INTERN ASSIGN CronEd.PR.Setpoint[57]:=(REAL_TO_WORD(CronEd.PR_TT*10))
rounded rectangle at (57,1063)-(88,1079): text "%.1f"; shows WORD_TO_REAL(CronEd.PR.Setpoint[58])/10; runs INTERN ASSIGN CronEd.PR.Setpoint[58]:=(REAL_TO_WORD(CronEd.PR_TT*10))
rounded rectangle at (57,1078)-(88,1094): text "%.1f"; shows WORD_TO_REAL(CronEd.PR.Setpoint[59])/10; runs INTERN ASSIGN CronEd.PR.Setpoint[59]:=(REAL_TO_WORD(CronEd.PR_TT*10))
button at (343,127)-(404,148): text "Load Hour"; toggles CronEd.PR_Load_Hour
button at (411,127)-(472,148): text "Save Hour"; toggles CronEd.PR_Save_Hour
group at (20,498)-(52,647)
  rectangle at (0,0)-(31,16): text "m20"
  rectangle at (0,15)-(31,31): text "m21"
  rectangle at (0,30)-(31,46): text "m22"
  rectangle at (0,45)-(31,61): text "m23"
  rectangle at (0,59)-(31,75): text "m24"
  rectangle at (0,74)-(31,90): text "m25"
  rectangle at (0,89)-(31,105): text "m26"
  rectangle at (0,104)-(31,120): text "m27"
  rectangle at (1,118)-(32,134): text "m28"
  rectangle at (1,133)-(32,149): text "m29"
group at (21,646)-(52,795)
  rectangle at (0,0)-(31,16): text "m30"
  rectangle at (0,15)-(31,31): text "m31"
  rectangle at (0,29)-(31,45): text "m32"
  rectangle at (0,44)-(31,60): text "m33"
  rectangle at (0,59)-(31,75): text "m34"
  rectangle at (0,74)-(31,90): text "m35"
  rectangle at (0,89)-(31,105): text "m36"
  rectangle at (0,104)-(31,120): text "m37"
  rectangle at (0,118)-(31,134): text "m38"
  rectangle at (0,133)-(31,149): text "m39"
group at (21,794)-(52,946)
  rectangle at (0,0)-(31,16): text "m40"
  rectangle at (0,15)-(31,31): text "m41"
  rectangle at (0,30)-(31,46): text "m42"
  rectangle at (0,45)-(31,61): text "m43"
  rectangle at (0,60)-(31,76): text "m44"
  rectangle at (0,75)-(31,91): text "m45"
  rectangle at (0,90)-(31,106): text "m46"
  rectangle at (0,105)-(31,121): text "m47"
  rectangle at (0,121)-(31,137): text "m48"
  rectangle at (0,136)-(31,152): text "m49"
group at (21,945)-(52,1097)
  rectangle at (0,0)-(31,16): text "m50"
  rectangle at (0,15)-(31,31): text "m51"
  rectangle at (0,30)-(31,46): text "m52"
  rectangle at (0,45)-(31,61): text "m53"
  rectangle at (0,60)-(31,76): text "m54"
  rectangle at (0,75)-(31,91): text "m55"
  rectangle at (0,90)-(31,106): text "m56"
  rectangle at (0,105)-(31,121): text "m57"
  rectangle at (0,121)-(31,137): text "m58"
  rectangle at (0,136)-(31,152): text "m59"
group at (574,174)-(605,326)
  rectangle at (0,0)-(31,16): text "m50"
  rectangle at (0,15)-(31,31): text "m51"
  rectangle at (0,30)-(31,46): text "m52"
  rectangle at (0,45)-(31,61): text "m53"
  rectangle at (0,60)-(31,76): text "m54"
  rectangle at (0,75)-(31,91): text "m55"
  rectangle at (0,90)-(31,106): text "m56"
  rectangle at (0,105)-(31,121): text "m57"
  rectangle at (0,121)-(31,137): text "m58"
  rectangle at (0,136)-(31,152): text "m59"
rounded rectangle at (615,173)-(646,189): text "%.1f"; shows WORD_TO_REAL(CronEd.PR_Minutes[50]/10); runs INTERN ASSIGN CronEd.PR_Minutes[50]:=(REAL_TO_WORD(CronEd.PR_TT*10))
rounded rectangle at (615,188)-(646,204): text "%.1f"; shows WORD_TO_REAL(CronEd.PR_Minutes[51]/10); runs INTERN ASSIGN CronEd.PR_Minutes[51]:=(REAL_TO_WORD(CronEd.PR_TT*10))
rounded rectangle at (615,203)-(646,219): text "%.1f"; shows WORD_TO_REAL(CronEd.PR_Minutes[52]/10); runs INTERN ASSIGN CronEd.PR_Minutes[52]:=(REAL_TO_WORD(CronEd.PR_TT*10))
rounded rectangle at (615,218)-(646,234): text "%.1f"; shows WORD_TO_REAL(CronEd.PR_Minutes[53]/10); runs INTERN ASSIGN CronEd.PR_Minutes[53]:=(REAL_TO_WORD(CronEd.PR_TT*10))
rounded rectangle at (615,233)-(646,249): text "%.1f"; shows WORD_TO_REAL(CronEd.PR_Minutes[54]/10); runs INTERN ASSIGN CronEd.PR_Minutes[54]:=(REAL_TO_WORD(CronEd.PR_TT*10))
rounded rectangle at (615,248)-(646,264): text "%.1f"; shows WORD_TO_REAL(CronEd.PR_Minutes[55]/10); runs INTERN ASSIGN CronEd.PR_Minutes[55]:=(REAL_TO_WORD(CronEd.PR_TT*10))
rounded rectangle at (615,263)-(646,279): text "%.1f"; shows WORD_TO_REAL(CronEd.PR_Minutes[56]/10); runs INTERN ASSIGN CronEd.PR_Minutes[56]:=(REAL_TO_WORD(CronEd.PR_TT*10))
rounded rectangle at (615,278)-(646,294): text "%.1f"; shows WORD_TO_REAL(CronEd.PR_Minutes[57]/10); runs INTERN ASSIGN CronEd.PR_Minutes[57]:=(REAL_TO_WORD(CronEd.PR_TT*10))
rounded rectangle at (615,293)-(646,309): text "%.1f"; shows WORD_TO_REAL(CronEd.PR_Minutes[58]/10); runs INTERN ASSIGN CronEd.PR_Minutes[58]:=(REAL_TO_WORD(CronEd.PR_TT*10))
rounded rectangle at (615,308)-(646,324): text "%.1f"; shows WORD_TO_REAL(CronEd.PR_Minutes[59]/10); runs INTERN ASSIGN CronEd.PR_Minutes[59]:=(REAL_TO_WORD(CronEd.PR_TT*10))
rounded rectangle at (533,173)-(564,189): text "%.1f"; shows WORD_TO_REAL(CronEd.PR_Minutes[40]/10); runs INTERN ASSIGN CronEd.PR_Minutes[40]:=(REAL_TO_WORD(CronEd.PR_TT*10))
rounded rectangle at (533,188)-(564,204): text "%.1f"; shows WORD_TO_REAL(CronEd.PR_Minutes[41]/10); runs INTERN ASSIGN CronEd.PR_Minutes[41]:=(REAL_TO_WORD(CronEd.PR_TT*10))
rounded rectangle at (533,203)-(564,219): text "%.1f"; shows WORD_TO_REAL(CronEd.PR_Minutes[42]/10); runs INTERN ASSIGN CronEd.PR_Minutes[42]:=(REAL_TO_WORD(CronEd.PR_TT*10))
rounded rectangle at (533,218)-(564,234): text "%.1f"; shows WORD_TO_REAL(CronEd.PR_Minutes[43]/10); runs INTERN ASSIGN CronEd.PR_Minutes[43]:=(REAL_TO_WORD(CronEd.PR_TT*10))
rounded rectangle at (533,233)-(564,249): text "%.1f"; shows WORD_TO_REAL(CronEd.PR_Minutes[44]/10); runs INTERN ASSIGN CronEd.PR_Minutes[44]:=(REAL_TO_WORD(CronEd.PR_TT*10))
rounded rectangle at (533,248)-(564,264): text "%.1f"; shows WORD_TO_REAL(CronEd.PR_Minutes[45]/10); runs INTERN ASSIGN CronEd.PR_Minutes[45]:=(REAL_TO_WORD(CronEd.PR_TT*10))
rounded rectangle at (533,263)-(564,279): text "%.1f"; shows WORD_TO_REAL(CronEd.PR_Minutes[46]/10); runs INTERN ASSIGN CronEd.PR_Minutes[46]:=(REAL_TO_WORD(CronEd.PR_TT*10))
rounded rectangle at (533,278)-(564,294): text "%.1f"; shows WORD_TO_REAL(CronEd.PR_Minutes[47]/10); runs INTERN ASSIGN CronEd.PR_Minutes[47]:=(REAL_TO_WORD(CronEd.PR_TT*10))
rounded rectangle at (533,293)-(564,309): text "%.1f"; shows WORD_TO_REAL(CronEd.PR_Minutes[48]/10); runs INTERN ASSIGN CronEd.PR_Minutes[48]:=(REAL_TO_WORD(CronEd.PR_TT*10))
rounded rectangle at (533,308)-(564,324): text "%.1f"; shows WORD_TO_REAL(CronEd.PR_Minutes[49]/10); runs INTERN ASSIGN CronEd.PR_Minutes[49]:=(REAL_TO_WORD(CronEd.PR_TT*10))
group at (493,173)-(524,325)
  rectangle at (0,0)-(31,16): text "m40"
  rectangle at (0,15)-(31,31): text "m41"
  rectangle at (0,30)-(31,46): text "m42"
  rectangle at (0,45)-(31,61): text "m43"
  rectangle at (0,60)-(31,76): text "m44"
  rectangle at (0,75)-(31,91): text "m45"
  rectangle at (0,90)-(31,106): text "m46"
  rectangle at (0,105)-(31,121): text "m47"
  rectangle at (0,121)-(31,137): text "m48"
  rectangle at (0,136)-(31,152): text "m49"
rounded rectangle at (453,173)-(484,189): text "%.1f"; shows WORD_TO_REAL(CronEd.PR_Minutes[30]/10); runs INTERN ASSIGN CronEd.PR_Minutes[30]:=(REAL_TO_WORD(CronEd.PR_TT*10))
rounded rectangle at (453,188)-(484,204): text "%.1f"; shows WORD_TO_REAL(CronEd.PR_Minutes[31]/10); runs INTERN ASSIGN CronEd.PR_Minutes[31]:=(REAL_TO_WORD(CronEd.PR_TT*10))
rounded rectangle at (453,203)-(484,219): text "%.1f"; shows WORD_TO_REAL(CronEd.PR_Minutes[32]/10); runs INTERN ASSIGN CronEd.PR_Minutes[32]:=(REAL_TO_WORD(CronEd.PR_TT*10))
rounded rectangle at (453,218)-(484,234): text "%.1f"; shows WORD_TO_REAL(CronEd.PR_Minutes[33]/10); runs INTERN ASSIGN CronEd.PR_Minutes[33]:=(REAL_TO_WORD(CronEd.PR_TT*10))
rounded rectangle at (453,233)-(484,249): text "%.1f"; shows WORD_TO_REAL(CronEd.PR_Minutes[34]/10); runs INTERN ASSIGN CronEd.PR_Minutes[34]:=(REAL_TO_WORD(CronEd.PR_TT*10))
rounded rectangle at (453,248)-(484,264): text "%.1f"; shows WORD_TO_REAL(CronEd.PR_Minutes[35]/10); runs INTERN ASSIGN CronEd.PR_Minutes[35]:=(REAL_TO_WORD(CronEd.PR_TT*10))
rounded rectangle at (453,263)-(484,279): text "%.1f"; shows WORD_TO_REAL(CronEd.PR_Minutes[36]/10); runs INTERN ASSIGN CronEd.PR_Minutes[36]:=(REAL_TO_WORD(CronEd.PR_TT*10))
rounded rectangle at (453,278)-(484,294): text "%.1f"; shows WORD_TO_REAL(CronEd.PR_Minutes[37]/10); runs INTERN ASSIGN CronEd.PR_Minutes[37]:=(REAL_TO_WORD(CronEd.PR_TT*10))
rounded rectangle at (453,293)-(484,309): text "%.1f"; shows WORD_TO_REAL(CronEd.PR_Minutes[38]/10); runs INTERN ASSIGN CronEd.PR_Minutes[38]:=(REAL_TO_WORD(CronEd.PR_TT*10))
rounded rectangle at (453,308)-(484,324): text "%.1f"; shows WORD_TO_REAL(CronEd.PR_Minutes[39]/10); runs INTERN ASSIGN CronEd.PR_Minutes[39]:=(REAL_TO_WORD(CronEd.PR_TT*10))
group at (413,175)-(444,324)
  rectangle at (0,0)-(31,16): text "m30"
  rectangle at (0,15)-(31,31): text "m31"
  rectangle at (0,29)-(31,45): text "m32"
  rectangle at (0,44)-(31,60): text "m33"
  rectangle at (0,59)-(31,75): text "m34"
  rectangle at (0,74)-(31,90): text "m35"
  rectangle at (0,89)-(31,105): text "m36"
  rectangle at (0,104)-(31,120): text "m37"
  rectangle at (0,118)-(31,134): text "m38"
  rectangle at (0,133)-(31,149): text "m39"
group at (336,174)-(367,323)
  rectangle at (0,0)-(31,16): text "m20"
  rectangle at (0,15)-(31,31): text "m21"
  rectangle at (0,30)-(31,46): text "m22"
  rectangle at (0,45)-(31,61): text "m23"
  rectangle at (0,59)-(31,75): text "m24"
  rectangle at (0,74)-(31,90): text "m25"
  rectangle at (0,89)-(31,105): text "m26"
  rectangle at (0,104)-(31,120): text "m27"
  rectangle at (0,118)-(31,134): text "m28"
  rectangle at (0,133)-(31,149): text "m29"
rounded rectangle at (375,173)-(406,189): text "%.1f"; shows WORD_TO_REAL(CronEd.PR_Minutes[20]/10); runs INTERN ASSIGN CronEd.PR_Minutes[20]:=(REAL_TO_WORD(CronEd.PR_TT*10))
rounded rectangle at (375,188)-(406,204): text "%.1f"; shows WORD_TO_REAL(CronEd.PR_Minutes[21]/10); runs INTERN ASSIGN CronEd.PR_Minutes[21]:=(REAL_TO_WORD(CronEd.PR_TT*10))
rounded rectangle at (375,203)-(406,219): text "%.1f"; shows WORD_TO_REAL(CronEd.PR_Minutes[22]/10); runs INTERN ASSIGN CronEd.PR_Minutes[22]:=(REAL_TO_WORD(CronEd.PR_TT*10))
rounded rectangle at (375,218)-(406,234): text "%.1f"; shows WORD_TO_REAL(CronEd.PR_Minutes[23]/10); runs INTERN ASSIGN CronEd.PR_Minutes[23]:=(REAL_TO_WORD(CronEd.PR_TT*10))
rounded rectangle at (375,233)-(406,249): text "%.1f"; shows WORD_TO_REAL(CronEd.PR_Minutes[24]/10); runs INTERN ASSIGN CronEd.PR_Minutes[24]:=(REAL_TO_WORD(CronEd.PR_TT*10))
rounded rectangle at (375,248)-(406,264): text "%.1f"; shows WORD_TO_REAL(CronEd.PR_Minutes[25]/10); runs INTERN ASSIGN CronEd.PR_Minutes[25]:=(REAL_TO_WORD(CronEd.PR_TT*10))
rounded rectangle at (375,263)-(406,279): text "%.1f"; shows WORD_TO_REAL(CronEd.PR_Minutes[26]/10); runs INTERN ASSIGN CronEd.PR_Minutes[26]:=(REAL_TO_WORD(CronEd.PR_TT*10))
rounded rectangle at (375,278)-(406,294): text "%.1f"; shows WORD_TO_REAL(CronEd.PR_Minutes[27]/10); runs INTERN ASSIGN CronEd.PR_Minutes[27]:=(REAL_TO_WORD(CronEd.PR_TT*10))
rounded rectangle at (375,293)-(406,309): text "%.1f"; shows WORD_TO_REAL(CronEd.PR_Minutes[28]/10); runs INTERN ASSIGN CronEd.PR_Minutes[28]:=(REAL_TO_WORD(CronEd.PR_TT*10))
rounded rectangle at (375,308)-(406,324): text "%.1f"; shows WORD_TO_REAL(CronEd.PR_Minutes[29]/10); runs INTERN ASSIGN CronEd.PR_Minutes[29]:=(REAL_TO_WORD(CronEd.PR_TT*10))
rounded rectangle at (296,173)-(327,189): text "%.1f"; shows WORD_TO_REAL(CronEd.PR_Minutes[10]/10); runs INTERN ASSIGN CronEd.PR_Minutes[10]:=(REAL_TO_WORD(CronEd.PR_TT*10))
rounded rectangle at (296,188)-(327,204): text "%.1f"; shows WORD_TO_REAL(CronEd.PR_Minutes[11]/10); runs INTERN ASSIGN CronEd.PR_Minutes[11]:=(REAL_TO_WORD(CronEd.PR_TT*10))
rounded rectangle at (296,203)-(327,219): text "%.1f"; shows WORD_TO_REAL(CronEd.PR_Minutes[12]/10); runs INTERN ASSIGN CronEd.PR_Minutes[12]:=(REAL_TO_WORD(CronEd.PR_TT*10))
rounded rectangle at (296,218)-(327,234): text "%.1f"; shows WORD_TO_REAL(CronEd.PR_Minutes[13]/10); runs INTERN ASSIGN CronEd.PR_Minutes[13]:=(REAL_TO_WORD(CronEd.PR_TT*10))
rounded rectangle at (296,233)-(327,249): text "%.1f"; shows WORD_TO_REAL(CronEd.PR_Minutes[14]/10); runs INTERN ASSIGN CronEd.PR_Minutes[14]:=(REAL_TO_WORD(CronEd.PR_TT*10))
rounded rectangle at (296,248)-(327,264): text "%.1f"; shows WORD_TO_REAL(CronEd.PR_Minutes[15]/10); runs INTERN ASSIGN CronEd.PR_Minutes[15]:=(REAL_TO_WORD(CronEd.PR_TT*10))
rounded rectangle at (296,263)-(327,279): text "%.1f"; shows WORD_TO_REAL(CronEd.PR_Minutes[16]/10); runs INTERN ASSIGN CronEd.PR_Minutes[16]:=(REAL_TO_WORD(CronEd.PR_TT*10))
rounded rectangle at (296,278)-(327,294): text "%.1f"; shows WORD_TO_REAL(CronEd.PR_Minutes[17]/10); runs INTERN ASSIGN CronEd.PR_Minutes[17]:=(REAL_TO_WORD(CronEd.PR_TT*10))
rounded rectangle at (296,293)-(327,309): text "%.1f"; shows WORD_TO_REAL(CronEd.PR_Minutes[18]/10); runs INTERN ASSIGN CronEd.PR_Minutes[18]:=(REAL_TO_WORD(CronEd.PR_TT*10))
rounded rectangle at (296,308)-(327,324): text "%.1f"; shows WORD_TO_REAL(CronEd.PR_Minutes[19]/10); runs INTERN ASSIGN CronEd.PR_Minutes[19]:=(REAL_TO_WORD(CronEd.PR_TT*10))
group at (257,174)-(288,323)
  rectangle at (0,0)-(31,16): text "m10"
  rectangle at (0,15)-(31,31): text "m11"
  rectangle at (0,29)-(31,45): text "m12"
  rectangle at (0,44)-(31,60): text "m13"
  rectangle at (0,59)-(31,75): text "m14"
  rectangle at (0,74)-(31,90): text "m15"
  rectangle at (0,88)-(31,104): text "m16"
  rectangle at (0,103)-(31,119): text "m17"
  rectangle at (0,118)-(31,134): text "m18"
  rectangle at (0,133)-(31,149): text "m19"
rounded rectangle at (220,173)-(251,189): text "%.1f"; shows WORD_TO_REAL(CronEd.PR_Minutes[0]/10); runs INTERN ASSIGN CronEd.PR_Minutes[0]:=(REAL_TO_WORD(CronEd.PR_TT*10))
rounded rectangle at (220,188)-(251,204): text "%.1f"; shows WORD_TO_REAL(CronEd.PR_Minutes[1]/10); runs INTERN ASSIGN CronEd.PR_Minutes[1]:=(REAL_TO_WORD(CronEd.PR_TT*10))
rounded rectangle at (220,203)-(251,219): text "%.1f"; shows WORD_TO_REAL(CronEd.PR_Minutes[2]/10); runs INTERN ASSIGN CronEd.PR_Minutes[2]:=(REAL_TO_WORD(CronEd.PR_TT*10))
rounded rectangle at (220,218)-(251,234): text "%.1f"; shows WORD_TO_REAL(CronEd.PR_Minutes[3]/10); runs INTERN ASSIGN CronEd.PR_Minutes[3]:=(REAL_TO_WORD(CronEd.PR_TT*10))
rounded rectangle at (220,233)-(251,249): text "%.1f"; shows WORD_TO_REAL(CronEd.PR_Minutes[4]/10); runs INTERN ASSIGN CronEd.PR_Minutes[4]:=(REAL_TO_WORD(CronEd.PR_TT*10))
rounded rectangle at (220,248)-(251,264): text "%.1f"; shows WORD_TO_REAL(CronEd.PR_Minutes[5]/10); runs INTERN ASSIGN CronEd.PR_Minutes[5]:=(REAL_TO_WORD(CronEd.PR_TT*10))
rounded rectangle at (220,263)-(251,279): text "%.1f"; shows WORD_TO_REAL(CronEd.PR_Minutes[6]/10); runs INTERN ASSIGN CronEd.PR_Minutes[6]:=(REAL_TO_WORD(CronEd.PR_TT*10))
rounded rectangle at (220,278)-(251,294): text "%.1f"; shows WORD_TO_REAL(CronEd.PR_Minutes[7]/10); runs INTERN ASSIGN CronEd.PR_Minutes[7]:=(REAL_TO_WORD(CronEd.PR_TT*10))
rounded rectangle at (220,293)-(251,309): text "%.1f"; shows WORD_TO_REAL(CronEd.PR_Minutes[8]/10); runs INTERN ASSIGN CronEd.PR_Minutes[8]:=(REAL_TO_WORD(CronEd.PR_TT*10))
rounded rectangle at (220,308)-(251,324): text "%.1f"; shows WORD_TO_REAL(CronEd.PR_Minutes[9]/10); runs INTERN ASSIGN CronEd.PR_Minutes[9]:=(REAL_TO_WORD(CronEd.PR_TT*10))
group at (182,174)-(213,323)
  rectangle at (0,0)-(31,16): text "m00"
  rectangle at (0,15)-(31,31): text "m01"
  rectangle at (0,30)-(31,46): text "m02"
  rectangle at (0,45)-(31,61): text "m03"
  rectangle at (0,59)-(31,75): text "m04"
  rectangle at (0,74)-(31,90): text "m05"
  rectangle at (0,89)-(31,105): text "m06"
  rectangle at (0,104)-(31,120): text "m07"
  rectangle at (0,118)-(31,134): text "m08"
  rectangle at (0,133)-(31,149): text "m09"
2 more shapes without text or variables
1 elements of other kinds (tables, trends, ...) not read
*)
